// TwinCAT 3 PLC project mobject_core
// Title: mobject-core
// Company: mobject
// Author: mobject dev team
// ProjectVersion: 0.10.0
// ProgramVersion: 3.1.4026.22
// libraries:
//   Tc2_Standard, * (Beckhoff Automation GmbH)
//   Tc2_System, * (Beckhoff Automation GmbH)
//   Tc2_Utilities, * (Beckhoff Automation GmbH)
//   Tc3_JsonXml, * (Beckhoff Automation GmbH)
// project tree:
//   mobject-collections/Dictionary/ Dictionary.TcPOU
//   mobject-collections/Interfaces/Collections/Events/ I_CollectionChangedEvent.TcIO, I_CollectionDisposedEvent.TcIO
//   mobject-collections/Interfaces/Collections/ I_Collection.TcIO (not stored), I_LinkedList.TcIO (not stored), I_List.TcIO, I_Queue.TcIO, I_Stack.TcIO (not stored)
//   mobject-collections/Interfaces/Collections/Nodes/ I_CollectionNode.TcIO, I_LinkedListNode.TcIO, I_ListNode.TcIO
//   mobject-collections/Interfaces/KeyValueCollections/Events/ I_KeyValueCollectionChangedEvent.TcIO, I_KeyValueCollectionDisposedEvent.TcIO
//   mobject-collections/Interfaces/KeyValueCollections/ I_Dictionary.TcIO, I_KeyValueCollection.TcIO
//   mobject-collections/Interfaces/KeyValueCollections/Nodes/ I_DictionaryTreeNode.TcIO (not stored), I_OrderedDictionaryTreeNode.TcIO (not stored)
//   mobject-collections/LinkedList/ LinkedList.TcPOU (not stored)
//   mobject-collections/OrderedDictionary/ OrderedDictionary.TcPOU
//   mobject-collections/Queue/ Queue.TcPOU
//   mobject-collections/Stack/ Stack.TcPOU (not stored)
//   mobject-collections/_Internal/Dictionary/Enumerator/ DictionaryForwardEnumerator.TcPOU (not stored)
//   mobject-collections/_Internal/Dictionary/Node/ DictionaryTreeNode.TcPOU (not stored)
//   mobject-collections/_Internal/Events/Collection/ CollectionChangedEvent.TcPOU, CollectionDisposedEvent.TcPOU, CollectionEvent.TcPOU
//   mobject-collections/_Internal/Events/KeyValueCollection/ KeyValueCollectionChangedEvent.TcPOU (not stored), KeyValueCollectionDisposedEvent.TcPOU (not stored), KeyValueCollectionEvent.TcPOU (not stored)
//   mobject-collections/_Internal/LinkedList/Enumerator/ LinkedListForwardEnumerator.TcPOU (not stored)
//   mobject-collections/_Internal/LinkedList/Node/ LinkedListNode.TcPOU (not stored)
//   mobject-collections/_Internal/OrderedDictionary/Enumerator/ OrderedDictionaryForwardEnumerator.TcPOU
//   mobject-collections/_Internal/OrderedDictionary/Node/ OrderedDictionaryTreeNode.TcPOU
//   mobject-commands/AsyncCommand/ AsyncCommand.TcPOU
//   mobject-commands/AsyncCommand/Interface/ I_AsyncCommand.TcIO (not stored)
//   mobject-commands/AsyncCommand/Runners/ SingleAsyncCommandRunner.TcPOU
//   mobject-commands/Command/Interface/ I_Command.TcIO (not stored)
//   mobject-commands/_Internal/AsyncCommandStateMachine/ AsyncCommandStateMachine.TcPOU (not stored), I_AsyncCommandStateControl.TcIO
//   mobject-constants/ DatatypeLimits.TcGVL (not stored)
//   mobject-converters/Converters/BOOL_TO_/ TryConvert_BOOL_TO_BOOL.TcPOU, TryConvert_BOOL_TO_BYTE.TcPOU (not stored), TryConvert_BOOL_TO_DATE.TcPOU (not stored), TryConvert_BOOL_TO_Destination.TcPOU (not stored), TryConvert_BOOL_TO_DINT.TcPOU (not stored), TryConvert_BOOL_TO_DT.TcPOU, TryConvert_BOOL_TO_DWORD.TcPOU, TryConvert_BOOL_TO_INT.TcPOU (not stored), TryConvert_BOOL_TO_LINT.TcPOU (not stored), TryConvert_BOOL_TO_LREAL.TcPOU, TryConvert_BOOL_TO_LWORD.TcPOU, TryConvert_BOOL_TO_REAL.TcPOU (not stored), TryConvert_BOOL_TO_SINT.TcPOU, TryConvert_BOOL_TO_STRING.TcPOU, TryConvert_BOOL_TO_TIME.TcPOU, TryConvert_BOOL_TO_TOD.TcPOU, TryConvert_BOOL_TO_UDINT.TcPOU (not stored), TryConvert_BOOL_TO_UINT.TcPOU (not stored), TryConvert_BOOL_TO_ULINT.TcPOU (not stored), TryConvert_BOOL_TO_USINT.TcPOU (not stored), TryConvert_BOOL_TO_WORD.TcPOU
//   mobject-converters/Converters/BYTE_TO_/ TryConvert_BYTE_TO_BOOL.TcPOU (not stored), TryConvert_BYTE_TO_BYTE.TcPOU, TryConvert_BYTE_TO_DATE.TcPOU (not stored), TryConvert_BYTE_TO_Destination.TcPOU, TryConvert_BYTE_TO_DINT.TcPOU (not stored), TryConvert_BYTE_TO_DT.TcPOU, TryConvert_BYTE_TO_DWORD.TcPOU (not stored), TryConvert_BYTE_TO_INT.TcPOU (not stored), TryConvert_BYTE_TO_LINT.TcPOU, TryConvert_BYTE_TO_LREAL.TcPOU, TryConvert_BYTE_TO_LWORD.TcPOU, TryConvert_BYTE_TO_REAL.TcPOU (not stored), TryConvert_BYTE_TO_SINT.TcPOU (not stored), TryConvert_BYTE_TO_STRING.TcPOU (not stored), TryConvert_BYTE_TO_TIME.TcPOU (not stored), TryConvert_BYTE_TO_TOD.TcPOU (not stored), TryConvert_BYTE_TO_UDINT.TcPOU, TryConvert_BYTE_TO_UINT.TcPOU, TryConvert_BYTE_TO_ULINT.TcPOU (not stored), TryConvert_BYTE_TO_USINT.TcPOU (not stored), TryConvert_BYTE_TO_WORD.TcPOU (not stored)
//   mobject-converters/Converters/DATE_TO_/ TryConvert_DATE_TO_BOOL.TcPOU, TryConvert_DATE_TO_BYTE.TcPOU, TryConvert_DATE_TO_DATE.TcPOU (not stored), TryConvert_DATE_TO_Destination.TcPOU, TryConvert_DATE_TO_DINT.TcPOU, TryConvert_DATE_TO_DT.TcPOU (not stored), TryConvert_DATE_TO_DWORD.TcPOU (not stored), TryConvert_DATE_TO_INT.TcPOU, TryConvert_DATE_TO_LINT.TcPOU, TryConvert_DATE_TO_LREAL.TcPOU (not stored), TryConvert_DATE_TO_LWORD.TcPOU (not stored), TryConvert_DATE_TO_REAL.TcPOU (not stored), TryConvert_DATE_TO_SINT.TcPOU, TryConvert_DATE_TO_STRING.TcPOU (not stored), TryConvert_DATE_TO_TIME.TcPOU, TryConvert_DATE_TO_TOD.TcPOU (not stored), TryConvert_DATE_TO_UDINT.TcPOU, TryConvert_DATE_TO_UINT.TcPOU (not stored), TryConvert_DATE_TO_ULINT.TcPOU (not stored), TryConvert_DATE_TO_USINT.TcPOU (not stored), TryConvert_DATE_TO_WORD.TcPOU (not stored)
//   mobject-converters/Converters/DINT_TO_/ TryConvert_DINT_TO_BOOL.TcPOU, TryConvert_DINT_TO_BYTE.TcPOU, TryConvert_DINT_TO_DATE.TcPOU (not stored), TryConvert_DINT_TO_Destination.TcPOU (not stored), TryConvert_DINT_TO_DINT.TcPOU (not stored), TryConvert_DINT_TO_DT.TcPOU, TryConvert_DINT_TO_DWORD.TcPOU, TryConvert_DINT_TO_INT.TcPOU, TryConvert_DINT_TO_LINT.TcPOU, TryConvert_DINT_TO_LREAL.TcPOU, TryConvert_DINT_TO_LWORD.TcPOU (not stored), TryConvert_DINT_TO_REAL.TcPOU (not stored), TryConvert_DINT_TO_SINT.TcPOU (not stored), TryConvert_DINT_TO_STRING.TcPOU, TryConvert_DINT_TO_TIME.TcPOU, TryConvert_DINT_TO_TOD.TcPOU, TryConvert_DINT_TO_UDINT.TcPOU (not stored), TryConvert_DINT_TO_UINT.TcPOU, TryConvert_DINT_TO_ULINT.TcPOU (not stored), TryConvert_DINT_TO_USINT.TcPOU, TryConvert_DINT_TO_WORD.TcPOU
//   mobject-converters/Converters/DT_TO_/ TryConvert_DT_TO_BOOL.TcPOU, TryConvert_DT_TO_BYTE.TcPOU, TryConvert_DT_TO_DATE.TcPOU (not stored), TryConvert_DT_TO_Destination.TcPOU (not stored), TryConvert_DT_TO_DINT.TcPOU, TryConvert_DT_TO_DT.TcPOU, TryConvert_DT_TO_DWORD.TcPOU, TryConvert_DT_TO_INT.TcPOU (not stored), TryConvert_DT_TO_LINT.TcPOU, TryConvert_DT_TO_LREAL.TcPOU (not stored), TryConvert_DT_TO_LWORD.TcPOU, TryConvert_DT_TO_REAL.TcPOU, TryConvert_DT_TO_SINT.TcPOU (not stored), TryConvert_DT_TO_STRING.TcPOU (not stored), TryConvert_DT_TO_TIME.TcPOU (not stored), TryConvert_DT_TO_TOD.TcPOU, TryConvert_DT_TO_UDINT.TcPOU (not stored), TryConvert_DT_TO_UINT.TcPOU, TryConvert_DT_TO_ULINT.TcPOU, TryConvert_DT_TO_USINT.TcPOU (not stored), TryConvert_DT_TO_WORD.TcPOU (not stored)
//   mobject-converters/Converters/DWORD_TO_/ TryConvert_DWORD_TO_BOOL.TcPOU (not stored), TryConvert_DWORD_TO_BYTE.TcPOU, TryConvert_DWORD_TO_DATE.TcPOU, TryConvert_DWORD_TO_Destination.TcPOU, TryConvert_DWORD_TO_DINT.TcPOU, TryConvert_DWORD_TO_DT.TcPOU, TryConvert_DWORD_TO_DWORD.TcPOU, TryConvert_DWORD_TO_INT.TcPOU, TryConvert_DWORD_TO_LINT.TcPOU, TryConvert_DWORD_TO_LREAL.TcPOU (not stored), TryConvert_DWORD_TO_LWORD.TcPOU, TryConvert_DWORD_TO_REAL.TcPOU, TryConvert_DWORD_TO_SINT.TcPOU (not stored), TryConvert_DWORD_TO_STRING.TcPOU, TryConvert_DWORD_TO_TIME.TcPOU, TryConvert_DWORD_TO_TOD.TcPOU, TryConvert_DWORD_TO_UDINT.TcPOU (not stored), TryConvert_DWORD_TO_UINT.TcPOU (not stored), TryConvert_DWORD_TO_ULINT.TcPOU (not stored), TryConvert_DWORD_TO_USINT.TcPOU, TryConvert_DWORD_TO_WORD.TcPOU (not stored)
//   mobject-converters/Converters/INT_TO_/ TryConvert_INT_TO_BOOL.TcPOU (not stored), TryConvert_INT_TO_BYTE.TcPOU (not stored), TryConvert_INT_TO_DATE.TcPOU, TryConvert_INT_TO_Destination.TcPOU (not stored), TryConvert_INT_TO_DINT.TcPOU (not stored), TryConvert_INT_TO_DT.TcPOU, TryConvert_INT_TO_DWORD.TcPOU (not stored), TryConvert_INT_TO_INT.TcPOU, TryConvert_INT_TO_LINT.TcPOU, TryConvert_INT_TO_LREAL.TcPOU (not stored), TryConvert_INT_TO_LWORD.TcPOU, TryConvert_INT_TO_REAL.TcPOU, TryConvert_INT_TO_SINT.TcPOU (not stored), TryConvert_INT_TO_STRING.TcPOU, TryConvert_INT_TO_TIME.TcPOU, TryConvert_INT_TO_TOD.TcPOU (not stored), TryConvert_INT_TO_UDINT.TcPOU, TryConvert_INT_TO_UINT.TcPOU (not stored), TryConvert_INT_TO_ULINT.TcPOU, TryConvert_INT_TO_USINT.TcPOU, TryConvert_INT_TO_WORD.TcPOU
//   mobject-converters/Converters/LINT_TO_/ TryConvert_LINT_TO_BOOL.TcPOU, TryConvert_LINT_TO_BYTE.TcPOU, TryConvert_LINT_TO_DATE.TcPOU, TryConvert_LINT_TO_Destination.TcPOU (not stored), TryConvert_LINT_TO_DINT.TcPOU, TryConvert_LINT_TO_DT.TcPOU, TryConvert_LINT_TO_DWORD.TcPOU, TryConvert_LINT_TO_INT.TcPOU, TryConvert_LINT_TO_LINT.TcPOU, TryConvert_LINT_TO_LREAL.TcPOU, TryConvert_LINT_TO_LWORD.TcPOU (not stored), TryConvert_LINT_TO_REAL.TcPOU (not stored), TryConvert_LINT_TO_SINT.TcPOU (not stored), TryConvert_LINT_TO_STRING.TcPOU, TryConvert_LINT_TO_TIME.TcPOU, TryConvert_LINT_TO_TOD.TcPOU, TryConvert_LINT_TO_UDINT.TcPOU (not stored), TryConvert_LINT_TO_UINT.TcPOU, TryConvert_LINT_TO_ULINT.TcPOU, TryConvert_LINT_TO_USINT.TcPOU, TryConvert_LINT_TO_WORD.TcPOU (not stored)
//   mobject-converters/Converters/LREAL_TO_/ TryConvert_LREAL_TO_BOOL.TcPOU, TryConvert_LREAL_TO_BYTE.TcPOU (not stored), TryConvert_LREAL_TO_DATE.TcPOU, TryConvert_LREAL_TO_Destination.TcPOU (not stored), TryConvert_LREAL_TO_DINT.TcPOU (not stored), TryConvert_LREAL_TO_DT.TcPOU, TryConvert_LREAL_TO_DWORD.TcPOU (not stored), TryConvert_LREAL_TO_INT.TcPOU, TryConvert_LREAL_TO_LINT.TcPOU (not stored), TryConvert_LREAL_TO_LREAL.TcPOU (not stored), TryConvert_LREAL_TO_LWORD.TcPOU (not stored), TryConvert_LREAL_TO_REAL.TcPOU (not stored), TryConvert_LREAL_TO_SINT.TcPOU (not stored), TryConvert_LREAL_TO_STRING.TcPOU, TryConvert_LREAL_TO_TIME.TcPOU (not stored), TryConvert_LREAL_TO_TOD.TcPOU (not stored), TryConvert_LREAL_TO_UDINT.TcPOU (not stored), TryConvert_LREAL_TO_UINT.TcPOU, TryConvert_LREAL_TO_ULINT.TcPOU, TryConvert_LREAL_TO_USINT.TcPOU, TryConvert_LREAL_TO_WORD.TcPOU
//   mobject-converters/Converters/LWORD_TO_/ TryConvert_LWORD_TO_BOOL.TcPOU (not stored), TryConvert_LWORD_TO_BYTE.TcPOU, TryConvert_LWORD_TO_DATE.TcPOU, TryConvert_LWORD_TO_Destination.TcPOU (not stored), TryConvert_LWORD_TO_DINT.TcPOU (not stored), TryConvert_LWORD_TO_DT.TcPOU (not stored), TryConvert_LWORD_TO_DWORD.TcPOU, TryConvert_LWORD_TO_INT.TcPOU, TryConvert_LWORD_TO_LINT.TcPOU (not stored), TryConvert_LWORD_TO_LREAL.TcPOU (not stored), TryConvert_LWORD_TO_LWORD.TcPOU, TryConvert_LWORD_TO_REAL.TcPOU, TryConvert_LWORD_TO_SINT.TcPOU, TryConvert_LWORD_TO_STRING.TcPOU (not stored), TryConvert_LWORD_TO_TIME.TcPOU (not stored), TryConvert_LWORD_TO_TOD.TcPOU (not stored), TryConvert_LWORD_TO_UDINT.TcPOU (not stored), TryConvert_LWORD_TO_UINT.TcPOU (not stored), TryConvert_LWORD_TO_ULINT.TcPOU, TryConvert_LWORD_TO_USINT.TcPOU (not stored), TryConvert_LWORD_TO_WORD.TcPOU
//   mobject-converters/Converters/REAL_TO_/ TryConvert_REAL_TO_BOOL.TcPOU (not stored), TryConvert_REAL_TO_BYTE.TcPOU (not stored), TryConvert_REAL_TO_DATE.TcPOU, TryConvert_REAL_TO_Destination.TcPOU (not stored), TryConvert_REAL_TO_DINT.TcPOU, TryConvert_REAL_TO_DT.TcPOU, TryConvert_REAL_TO_DWORD.TcPOU, TryConvert_REAL_TO_INT.TcPOU, TryConvert_REAL_TO_LINT.TcPOU, TryConvert_REAL_TO_LREAL.TcPOU (not stored), TryConvert_REAL_TO_LWORD.TcPOU (not stored), TryConvert_REAL_TO_REAL.TcPOU, TryConvert_REAL_TO_SINT.TcPOU, TryConvert_REAL_TO_STRING.TcPOU, TryConvert_REAL_TO_TIME.TcPOU, TryConvert_REAL_TO_TOD.TcPOU, TryConvert_REAL_TO_UDINT.TcPOU, TryConvert_REAL_TO_UINT.TcPOU, TryConvert_REAL_TO_ULINT.TcPOU, TryConvert_REAL_TO_USINT.TcPOU, TryConvert_REAL_TO_WORD.TcPOU
//   mobject-converters/Converters/SINT_TO_/ TryConvert_SINT_TO_BOOL.TcPOU (not stored), TryConvert_SINT_TO_BYTE.TcPOU, TryConvert_SINT_TO_DATE.TcPOU (not stored), TryConvert_SINT_TO_Destination.TcPOU (not stored), TryConvert_SINT_TO_DINT.TcPOU (not stored), TryConvert_SINT_TO_DT.TcPOU, TryConvert_SINT_TO_DWORD.TcPOU (not stored), TryConvert_SINT_TO_INT.TcPOU, TryConvert_SINT_TO_LINT.TcPOU, TryConvert_SINT_TO_LREAL.TcPOU, TryConvert_SINT_TO_LWORD.TcPOU (not stored), TryConvert_SINT_TO_REAL.TcPOU (not stored), TryConvert_SINT_TO_SINT.TcPOU (not stored), TryConvert_SINT_TO_STRING.TcPOU (not stored), TryConvert_SINT_TO_TIME.TcPOU (not stored), TryConvert_SINT_TO_TOD.TcPOU (not stored), TryConvert_SINT_TO_UDINT.TcPOU, TryConvert_SINT_TO_UINT.TcPOU, TryConvert_SINT_TO_ULINT.TcPOU, TryConvert_SINT_TO_USINT.TcPOU (not stored), TryConvert_SINT_TO_WORD.TcPOU (not stored)
//   mobject-converters/Converters/STRING_TO_/ TryConvert_STRING_TO_BOOL.TcPOU (not stored), TryConvert_STRING_TO_BYTE.TcPOU, TryConvert_STRING_TO_DATE.TcPOU, TryConvert_STRING_TO_Destination.TcPOU, TryConvert_STRING_TO_DINT.TcPOU, TryConvert_STRING_TO_DT.TcPOU (not stored), TryConvert_STRING_TO_DWORD.TcPOU, TryConvert_STRING_TO_INT.TcPOU (not stored), TryConvert_STRING_TO_LINT.TcPOU (not stored), TryConvert_STRING_TO_LREAL.TcPOU, TryConvert_STRING_TO_LWORD.TcPOU (not stored), TryConvert_STRING_TO_REAL.TcPOU, TryConvert_STRING_TO_SINT.TcPOU, TryConvert_STRING_TO_STRING.TcPOU, TryConvert_STRING_TO_TIME.TcPOU (not stored), TryConvert_STRING_TO_TOD.TcPOU, TryConvert_STRING_TO_UDINT.TcPOU (not stored), TryConvert_STRING_TO_UINT.TcPOU, TryConvert_STRING_TO_ULINT.TcPOU, TryConvert_STRING_TO_USINT.TcPOU, TryConvert_STRING_TO_WORD.TcPOU
//   mobject-converters/Converters/TIME_TO_/ TryConvert_TIME_TO_BOOL.TcPOU, TryConvert_TIME_TO_BYTE.TcPOU, TryConvert_TIME_TO_DATE.TcPOU (not stored), TryConvert_TIME_TO_Destination.TcPOU (not stored), TryConvert_TIME_TO_DINT.TcPOU, TryConvert_TIME_TO_DT.TcPOU (not stored), TryConvert_TIME_TO_DWORD.TcPOU, TryConvert_TIME_TO_INT.TcPOU, TryConvert_TIME_TO_LINT.TcPOU (not stored), TryConvert_TIME_TO_LREAL.TcPOU (not stored), TryConvert_TIME_TO_LWORD.TcPOU, TryConvert_TIME_TO_REAL.TcPOU, TryConvert_TIME_TO_SINT.TcPOU, TryConvert_TIME_TO_STRING.TcPOU, TryConvert_TIME_TO_TIME.TcPOU, TryConvert_TIME_TO_TOD.TcPOU (not stored), TryConvert_TIME_TO_UDINT.TcPOU, TryConvert_TIME_TO_UINT.TcPOU (not stored), TryConvert_TIME_TO_ULINT.TcPOU (not stored), TryConvert_TIME_TO_USINT.TcPOU, TryConvert_TIME_TO_WORD.TcPOU
//   mobject-converters/Converters/TOD_TO_/ TryConvert_TOD_TO_BOOL.TcPOU, TryConvert_TOD_TO_BYTE.TcPOU, TryConvert_TOD_TO_DATE.TcPOU (not stored), TryConvert_TOD_TO_Destination.TcPOU, TryConvert_TOD_TO_DINT.TcPOU (not stored), TryConvert_TOD_TO_DT.TcPOU (not stored), TryConvert_TOD_TO_DWORD.TcPOU (not stored), TryConvert_TOD_TO_INT.TcPOU, TryConvert_TOD_TO_LINT.TcPOU, TryConvert_TOD_TO_LREAL.TcPOU (not stored), TryConvert_TOD_TO_LWORD.TcPOU (not stored), TryConvert_TOD_TO_REAL.TcPOU, TryConvert_TOD_TO_SINT.TcPOU (not stored), TryConvert_TOD_TO_STRING.TcPOU (not stored), TryConvert_TOD_TO_TIME.TcPOU, TryConvert_TOD_TO_TOD.TcPOU (not stored), TryConvert_TOD_TO_UDINT.TcPOU (not stored), TryConvert_TOD_TO_UINT.TcPOU (not stored), TryConvert_TOD_TO_ULINT.TcPOU (not stored), TryConvert_TOD_TO_USINT.TcPOU, TryConvert_TOD_TO_WORD.TcPOU
//   mobject-converters/Converters/ TryConvert_Source_TO_Destination.TcPOU (not stored)
//   mobject-converters/Converters/UDINT_TO_/ TryConvert_UDINT_TO_BOOL.TcPOU, TryConvert_UDINT_TO_BYTE.TcPOU, TryConvert_UDINT_TO_DATE.TcPOU, TryConvert_UDINT_TO_Destination.TcPOU (not stored), TryConvert_UDINT_TO_DINT.TcPOU (not stored), TryConvert_UDINT_TO_DT.TcPOU (not stored), TryConvert_UDINT_TO_DWORD.TcPOU, TryConvert_UDINT_TO_INT.TcPOU, TryConvert_UDINT_TO_LINT.TcPOU (not stored), TryConvert_UDINT_TO_LREAL.TcPOU, TryConvert_UDINT_TO_LWORD.TcPOU, TryConvert_UDINT_TO_REAL.TcPOU, TryConvert_UDINT_TO_SINT.TcPOU (not stored), TryConvert_UDINT_TO_STRING.TcPOU, TryConvert_UDINT_TO_TIME.TcPOU (not stored), TryConvert_UDINT_TO_TOD.TcPOU (not stored), TryConvert_UDINT_TO_UDINT.TcPOU (not stored), TryConvert_UDINT_TO_UINT.TcPOU (not stored), TryConvert_UDINT_TO_ULINT.TcPOU (not stored), TryConvert_UDINT_TO_USINT.TcPOU, TryConvert_UDINT_TO_WORD.TcPOU
//   mobject-converters/Converters/UINT_TO_/ TryConvert_UINT_TO_BOOL.TcPOU, TryConvert_UINT_TO_BYTE.TcPOU (not stored), TryConvert_UINT_TO_DATE.TcPOU, TryConvert_UINT_TO_Destination.TcPOU, TryConvert_UINT_TO_DINT.TcPOU (not stored), TryConvert_UINT_TO_DT.TcPOU (not stored), TryConvert_UINT_TO_DWORD.TcPOU, TryConvert_UINT_TO_INT.TcPOU, TryConvert_UINT_TO_LINT.TcPOU, TryConvert_UINT_TO_LREAL.TcPOU, TryConvert_UINT_TO_LWORD.TcPOU (not stored), TryConvert_UINT_TO_REAL.TcPOU, TryConvert_UINT_TO_SINT.TcPOU, TryConvert_UINT_TO_STRING.TcPOU (not stored), TryConvert_UINT_TO_TIME.TcPOU, TryConvert_UINT_TO_TOD.TcPOU, TryConvert_UINT_TO_UDINT.TcPOU, TryConvert_UINT_TO_UINT.TcPOU, TryConvert_UINT_TO_ULINT.TcPOU (not stored), TryConvert_UINT_TO_USINT.TcPOU (not stored), TryConvert_UINT_TO_WORD.TcPOU (not stored)
//   mobject-converters/Converters/ULINT_TO_/ TryConvert_ULINT_TO_BOOL.TcPOU (not stored), TryConvert_ULINT_TO_BYTE.TcPOU, TryConvert_ULINT_TO_DATE.TcPOU, TryConvert_ULINT_TO_Destination.TcPOU, TryConvert_ULINT_TO_DINT.TcPOU (not stored), TryConvert_ULINT_TO_DT.TcPOU (not stored), TryConvert_ULINT_TO_DWORD.TcPOU, TryConvert_ULINT_TO_INT.TcPOU, TryConvert_ULINT_TO_LINT.TcPOU, TryConvert_ULINT_TO_LREAL.TcPOU, TryConvert_ULINT_TO_LWORD.TcPOU (not stored), TryConvert_ULINT_TO_REAL.TcPOU, TryConvert_ULINT_TO_SINT.TcPOU (not stored), TryConvert_ULINT_TO_STRING.TcPOU (not stored), TryConvert_ULINT_TO_TIME.TcPOU, TryConvert_ULINT_TO_TOD.TcPOU, TryConvert_ULINT_TO_UDINT.TcPOU (not stored), TryConvert_ULINT_TO_UINT.TcPOU, TryConvert_ULINT_TO_ULINT.TcPOU, TryConvert_ULINT_TO_USINT.TcPOU (not stored), TryConvert_ULINT_TO_WORD.TcPOU
//   mobject-converters/Converters/USINT_TO_/ TryConvert_USINT_TO_BOOL.TcPOU (not stored), TryConvert_USINT_TO_BYTE.TcPOU (not stored), TryConvert_USINT_TO_DATE.TcPOU, TryConvert_USINT_TO_Destination.TcPOU, TryConvert_USINT_TO_DINT.TcPOU (not stored), TryConvert_USINT_TO_DT.TcPOU (not stored), TryConvert_USINT_TO_DWORD.TcPOU, TryConvert_USINT_TO_INT.TcPOU (not stored), TryConvert_USINT_TO_LINT.TcPOU, TryConvert_USINT_TO_LREAL.TcPOU, TryConvert_USINT_TO_LWORD.TcPOU (not stored), TryConvert_USINT_TO_REAL.TcPOU, TryConvert_USINT_TO_SINT.TcPOU, TryConvert_USINT_TO_STRING.TcPOU, TryConvert_USINT_TO_TIME.TcPOU, TryConvert_USINT_TO_TOD.TcPOU (not stored), TryConvert_USINT_TO_UDINT.TcPOU, TryConvert_USINT_TO_UINT.TcPOU (not stored), TryConvert_USINT_TO_ULINT.TcPOU (not stored), TryConvert_USINT_TO_USINT.TcPOU, TryConvert_USINT_TO_WORD.TcPOU
//   mobject-converters/Converters/WORD_TO_/ TryConvert_WORD_TO_BOOL.TcPOU (not stored), TryConvert_WORD_TO_BYTE.TcPOU, TryConvert_WORD_TO_DATE.TcPOU, TryConvert_WORD_TO_Destination.TcPOU, TryConvert_WORD_TO_DINT.TcPOU, TryConvert_WORD_TO_DT.TcPOU (not stored), TryConvert_WORD_TO_DWORD.TcPOU, TryConvert_WORD_TO_INT.TcPOU, TryConvert_WORD_TO_LINT.TcPOU (not stored), TryConvert_WORD_TO_LREAL.TcPOU, TryConvert_WORD_TO_LWORD.TcPOU (not stored), TryConvert_WORD_TO_REAL.TcPOU (not stored), TryConvert_WORD_TO_SINT.TcPOU (not stored), TryConvert_WORD_TO_STRING.TcPOU, TryConvert_WORD_TO_TIME.TcPOU (not stored), TryConvert_WORD_TO_TOD.TcPOU, TryConvert_WORD_TO_UDINT.TcPOU, TryConvert_WORD_TO_UINT.TcPOU, TryConvert_WORD_TO_ULINT.TcPOU (not stored), TryConvert_WORD_TO_USINT.TcPOU (not stored), TryConvert_WORD_TO_WORD.TcPOU
//   mobject-datatypes/DatatypeOperations/Collection/ DatatypeOperations.TcPOU
//   mobject-datatypes/DatatypeOperations/Interface/ I_DatatypeOperation.TcIO (not stored)
//   mobject-datatypes/DatatypeOperations/ MemCopyOperation.TcPOU (not stored), SafeMemCopyOperation.TcPOU (not stored), WriteBitToBoolOperation.TcPOU, WriteBoolToBitOperation.TcPOU
//   mobject-datatypes/Datatypes/Base/ Datatypes.TcPOU (not stored)
//   mobject-datatypes/Datatypes/Events/ I_AliasDatatypeAddedEvent.TcIO (not stored), I_DatatypeAddedEvent.TcIO, I_EnumDatatypeAddedEvent.TcIO, I_InterfaceDatatypeAddedEvent.TcIO (not stored), I_StructuredDatatypeAddedEvent.TcIO (not stored), I_ArrayDatatypeAddedEvent.TcIO (not stored)
//   mobject-datatypes/Datatypes/Interface/ I_Datatypes.TcIO
//   mobject-datatypes/DatatypeVisitor/ I_DatatypeVisitor.TcIO
//   mobject-datatypes/Functions/ GetByteOffset.TcPOU (not stored)
//   mobject-datatypes/Primitive/Interfaces/ I_BIT.TcIO, I_BYTE.TcIO, I_ANY.TcIO, I_DINT.TcIO, I_DT.TcIO, I_DWORD.TcIO, I_INT.TcIO, I_LINT.TcIO, I_LREAL.TcIO, I_LWORD.TcIO, I_PVOID.TcIO, I_REAL.TcIO, I_REFERENCE_TO.TcIO, I_SINT.TcIO, I_TOD.TcIO, I_TIME_OF_DAY.TcIO, I_STRING.TcIO, I_BOOL.TcIO, I_UDINT.TcIO, I_UINT.TcIO, I_ULINT.TcIO, I_USINT.TcIO, I_WORD.TcIO
//   mobject-datatypes/Primitive/ _REFERENCE_TO.TcPOU, _NULL.TcPOU, _BIT.TcPOU, _BOOL.TcPOU, _ANY.TcPOU, _BYTE.TcPOU, _DINT.TcPOU, _DT.TcPOU, _DWORD.TcPOU, _INT.TcPOU, _LINT.TcPOU, _LREAL.TcPOU, _LWORD.TcPOU, _REAL.TcPOU, _SINT.TcPOU, _STRING.TcPOU, _TIME_OF_DAY.TcPOU, _TOD.TcPOU, _UDINT.TcPOU, _PVOID.TcPOU, _UINT.TcPOU, _ULINT.TcPOU, _USINT.TcPOU, _WORD.TcPOU
//   mobject-datatypes/_Internal/Datatype/ AliasDatatypeBase.TcPOU, ArrayDatatypeBase_2D.TcPOU (not stored), ArrayDatatypeBase_3D.TcPOU, DatatypeBase.TcPOU, EnumDatatypeBase.TcPOU, InterfaceDatatypeBase.TcPOU, NumericDatatypeBase.TcPOU (not stored), StructuredDatatypeBase.TcPOU, ArrayDatatypeBase_1D.TcPOU (not stored), UserDefinedDatatypeBase.TcPOU
//   mobject-datatypes/_Internal/Datatype/Interface/ I_AliasDatatype.TcIO, I_ArrayDatatype_1D.TcIO, I_ArrayDatatype_2D.TcIO (not stored), I_ArrayDatatype_3D.TcIO, I_Datatype.TcIO, I_EnumDatatype.TcIO, I_InterfaceDatatype.TcIO, I_NumericDatatype.TcIO (not stored), I_StructuredDatatype.TcIO, I_ArrayDatatype.TcIO, I_UserDefinedDatatype.TcIO
//   mobject-datatypes/_Internal/Errors/ UnknownEnumerationError.TcPOU (not stored)
//   mobject-datatypes/_Internal/Events/ AliasDatatypeAddedEvent.TcPOU (not stored), DatatypeAddedEvent.TcPOU, EnumDatatypeAddedEvent.TcPOU (not stored), InterfaceDatatypeAddedEvent.TcPOU, StructuredDatatypeAddedEvent.TcPOU, ArrayDatatypeAddedEvent.TcPOU (not stored)
//   mobject-datatypes/_Internal/StructureMembers/Host/ StructureMemberHost.TcPOU
//   mobject-datatypes/_Internal/StructureMembers/Interface/ I_HostStructureMembers.TcIO, I_StructureMembers.TcIO (not stored)
//   mobject-deserialization/DeserializationFeedback/ DeserializerFeedback.TcPOU
//   mobject-deserialization/Errors/CustomError/ CustomDeserializationFailedError.TcPOU (not stored)
//   mobject-deserialization/Errors/ DeserializationErrorFactory.TcPOU
//   mobject-deserialization/Errors/IncorrectType/ IncorrectKeyTypeDeserializationError.TcPOU, IncorrectTypeDeserializationError.TcPOU
//   mobject-deserialization/Errors/Invalid Index/ InvalidArrayIndexDeserializationError.TcPOU
//   mobject-deserialization/Errors/Invalid Key/ InvalidKeyDeserializationError.TcPOU (not stored)
//   mobject-deserialization/Errors/Missing Key/ MissingKeyDeserializationError.TcPOU
//   mobject-deserialization/GarbageCollector/ DeserializerGarbageCollector.TcPOU, I_DeserializerGarbageCollector.TcIO (not stored)
//   mobject-deserialization/Interfaces/ I_Deserializable.TcIO (not stored), I_Deserializer.TcIO, I_DeserializerArrayForwardEnumerator.TcIO, I_DeserializerFeedback.TcIO, I_DeserializerObjectForwardEnumerator.TcIO
//   mobject-errors/Errors/ Error.TcPOU (not stored), NullError.TcPOU
//   mobject-errors/Interfaces/ I_Error.TcIO, I_ErrorVisitor.TcIO
//   mobject-events/EventEmitter/ EventEmitter.TcPOU (not stored)
//   mobject-events/Interfaces/ I_Event.TcIO, I_EventEmitter.TcIO (not stored), I_EventHandler.TcIO (not stored), I_EventTarget.TcIO (not stored)
//   mobject-events/_Internal/EventHandlerItem/ EventHandlerItem.TcPOU, EventHandlerItemOnceOnly.TcPOU, I_EventHandlerItem.TcIO
//   mobject-disposable/Disposable/ Disposable.TcPOU (not stored)
//   mobject-disposable/Interfaces/ I_Disposable.TcIO (not stored)
//   mobject-enumerable/Interfaces/Enumerators/ I_ForwardEnumerator.TcIO, I_KeyValueForwardEnumerator.TcIO (not stored)
//   mobject-enumerable/Interfaces/ I_Enumerable.TcIO, I_KeyValueEnumerable.TcIO
//   mobject-json/JsonDeserializer/Events/ I_JsonDeserializerChangedEvent.TcIO (not stored), I_JsonDeserializerDisposedEvent.TcIO
//   mobject-json/JsonDeserializer/ I_JsonDeserializer.TcIO, JsonDeserializer.TcPOU
//   mobject-json/JsonDomParser/ JsonDomParser.TcPOU
//   mobject-json/JsonSerializer/ JsonSerializer.TcPOU
//   mobject-json/_Internal/Events/ JsonDeserializerChangedEvent.TcPOU, JsonDeserializerDisposedEvent.TcPOU (not stored), JsonDeserializerEvent.TcPOU
//   mobject-json/_Internal/JsonDeserializerForwardEnumerator/ JsonDeserializerArrayForwardEnumerator.TcPOU, JsonDeserializerNullArrayForwardEnumerator.TcPOU, JsonDeserializerNullObjectForwardEnumerator.TcPOU (not stored), JsonDeserializerObjectForwardEnumerator.TcPOU
//   mobject-json/_Internal/JsonDeserializerNode/ JsonDeserializerNode.TcPOU, JsonDeserializerNullNode.TcPOU
//   mobject-json/_Internal/JsonPathSyntaxParser/ JsonPathSyntaxParser.TcPOU
//   mobject-json/_Internal/JsonPathVisitor/ I_JsonPathVisitor.TcIO (not stored), JsonDomCreator.TcPOU, JsonDomNavigator.TcPOU (not stored)
//   mobject-serialization/Interfaces/ I_Serializable.TcIO, I_Serializer.TcIO
//   mobject-server/GVLs/ ServerConfiguration.TcGVL
//   mobject-server/RpcApi/ I_RpcApi.TcIO
//   mobject-server/RpcHandler/Examples/ AsyncConcatStringRpcHandler.TcPOU, ConcatStringRpcHandler.TcPOU
//   mobject-server/RpcHandler/ I_AsynchronousRpcHandler.TcIO, I_SynchronousRpcHandler.TcIO
//   mobject-server/RpcServer/ I_RpcServer.TcIO, RpcServer.TcPOU
//   mobject-server/_Internal/AsyncResponse/HeaderAccessor/ I_AsyncResponseHeaderAccessor.TcIO
//   mobject-server/_Internal/AsyncResponse/Manager/ AsyncResponseManager.TcPOU, I_AsyncResponseManager.TcIO
//   mobject-server/_Internal/AsyncResponse/Middleware/ AsyncResponseMiddleware.TcPOU
//   mobject-server/_Internal/AsyncResponse/Proxy/ AsyncResponseSessionDataProxy.TcPOU
//   mobject-server/_Internal/AsyncResponse/SessionData/ AsyncResponseSessionData.TcPOU, I_AsyncResponseSessionData.TcIO
//   mobject-server/_Internal/ChunkedRequests/ChunkedRequest/ ChunkedRequest.TcPOU
//   mobject-server/_Internal/ChunkedRequests/HeaderAccessor/ I_ChunkedRequestsHeaderAccessor.TcIO
//   mobject-server/_Internal/ChunkedRequests/Manager/ ChunkedRequestsManager.TcPOU, I_ChunkedRequestsManager.TcIO
//   mobject-server/_Internal/ChunkedRequests/Middleware/ ChunkedRequestsMiddleware.TcPOU
//   mobject-server/_Internal/ChunkedRequests/SessionData/ ChunkedRequestData.TcPOU, I_ChunkedRequestData.TcIO
//   mobject-server/_Internal/ChunkedResponses/HeaderAccessor/ I_ChunkedResponseHeaderAccessor.TcIO
//   mobject-server/_Internal/ChunkedResponses/Manager/ ChunkedResponseManager.TcPOU, I_ChunkedResponseManager.TcIO
//   mobject-server/_Internal/ChunkedResponses/Middleware/ ChunkedResponsesMiddleware.TcPOU
//   mobject-server/_Internal/ChunkedResponses/ServerResponse/ ChunkableServerResponse.TcPOU
//   mobject-server/_Internal/ChunkedResponses/SessionData/ ChunkedResponseData.TcPOU, I_ChunkedResponseData.TcIO
//   mobject-server/_Internal/Followup/Middleware/ ResponseIdGuardMiddleware.TcPOU
//   mobject-server/_Internal/HeaderAccessor/ HeaderAccessor.TcPOU
//   mobject-server/_Internal/Header/ Header.TcPOU, I_Header.TcIO
//   mobject-server/_Internal/Middleware/Base/ MiddlewareBase.TcPOU
//   mobject-server/_Internal/Middleware/Interface/ I_Middleware.TcIO
//   mobject-server/_Internal/Middleware/Stack/ MiddlewareStack.TcPOU
//   mobject-server/_Internal/Request/Interface/ I_Request.TcIO
//   mobject-server/_Internal/Request/ Request.TcPOU
//   mobject-server/_Internal/ResponseId/Interface/ I_ResponseIdGenerator.TcIO
//   mobject-server/_Internal/ResponseId/ SequentialResponseIdGenerator.TcPOU
//   mobject-server/_Internal/RPC/AsyncRpcCallQueue/ AsyncRpcCallQueue.TcPOU, I_AsyncRpcCallQueue.TcIO
//   mobject-server/_Internal/RPC/AsyncRpcCall/ AsyncRpcCall.TcPOU, I_AsyncRpcCall.TcIO
//   mobject-server/_Internal/RPC/Handlers/ AsynchronousRpcHandlers.TcPOU, I_AsynchronousRpcHandlers.TcIO, I_HostAsynchronousRpcHandlers.TcIO, I_HostSynchronousRpcHandlers.TcIO, I_SynchronousRpcHandlers.TcIO, SynchronousRpcHandlers.TcPOU
//   mobject-server/_Internal/RPC/HeaderAccessor/ I_RpcHeaderAccessor.TcIO
//   mobject-server/_Internal/RPC/Manager/ I_RpcManager.TcIO, RpcManager.TcPOU
//   mobject-server/_Internal/RPC/Middleware/ RpcMiddleware.TcPOU
//   mobject-server/_Internal/RPC/RegisteredRpcApis/ RegisteredRpcApis.TcPOU
//   mobject-server/_Internal/RPC/Response/Async/ AsynchronousRpcResponse.TcPOU, I_AsynchronousRpcResponse.TcIO
//   mobject-server/_Internal/RPC/Response/Factory/ AsynchronousRpcResponseFactory.TcPOU, I_AsynchronousRpcResponseFactory.TcIO
//   mobject-server/_Internal/RPC/Response/Sync/ I_SynchronousRpcResponse.TcIO, SynchronousRpcResponse.TcPOU
//   mobject-server/_Internal/ServerResponse/Data/ ResponseData.TcDUT
//   mobject-server/_Internal/ServerResponse/HeaderAccessor/ I_ServerResponseHeaderAccessor.TcIO
//   mobject-server/_Internal/ServerResponse/Interface/ I_ServerResponse.TcIO
//   mobject-server/_Internal/ServerResponse/ ServerResponse.TcPOU
//   mobject-server/_Internal/Sessions/HeaderAccessor/ I_SessionHeaderAccessor.TcIO
//   mobject-server/_Internal/Sessions/Manager/ I_SessionManager.TcIO, SessionManager.TcPOU
//   mobject-server/_Internal/Sessions/Middleware/ SessionsMiddleware.TcPOU
//   mobject-server/_Internal/Sessions/SessionData/ I_SessionData.TcIO
//   mobject-server/_Internal/Sessions/SessionId/ I_SessionIdGenerator.TcIO, SequentialSessionIdGenerator.TcPOU
//   mobject-server/_Internal/Sessions/Session/ I_Session.TcIO, Session.TcPOU
//   mobject-server/_Internal/Sessions/Storage/ I_SessionStorage.TcIO
//   mobject-server/_Internal/TimeStamp/ I_Timestamp.TcIO, SystemTimestamp.TcPOU

// ---- mobject-server/_Internal/ServerResponse/Data/ResponseData.TcDUT
TYPE ResponseData : 
STRUCT
	Header : STRING(ServerConfiguration.HEADER_STRING_SIZE);
	Payload : STRING(ServerConfiguration.PAYLOAD_STRING_SIZE);
END_STRUCT
END_TYPE

// ---- mobject-server/GVLs/ServerConfiguration.TcGVL
{attribute 'qualified_only'}
VAR_GLOBAL CONSTANT
	HEADER_STRING_SIZE : UDINT := 1024;
	PAYLOAD_STRING_SIZE : UDINT := 8000; // typically 1/8th of the Runtime Stack Size

	// Maximum time an asynchronous response may remain pending.
    // T#0S disables the deadline.
    PENDING_RESPONSE_MAX_AGE : TIME := T#60S;

    // Delay suggested to clients between asynchronous response polls.
    // Prevents clients continuously polling the PLC as fast as ADS allows.
    PENDING_RESPONSE_RETRY_DELAY_MS : UDINT := 20;
END_VAR

// ---- mobject-collections/Interfaces/Collections/Events/I_CollectionChangedEvent.TcIO
INTERFACE I_CollectionChangedEvent EXTENDS I_Event

PROPERTY PUBLIC Target : I_Collection
GET
END_GET
END_PROPERTY

END_INTERFACE

// ---- mobject-collections/Interfaces/Collections/Events/I_CollectionDisposedEvent.TcIO
INTERFACE I_CollectionDisposedEvent EXTENDS I_Event

PROPERTY PUBLIC Target : I_Collection
GET
END_GET
END_PROPERTY

END_INTERFACE

// ---- mobject-collections/Interfaces/Collections/I_List.TcIO
INTERFACE I_List EXTENDS I_Collection

PROPERTY PUBLIC Capacity : DINT
GET
END_GET
END_PROPERTY

METHOD PUBLIC GetIndexOf : DINT
VAR_INPUT
	Item : ANY;
END_VAR
END_METHOD

METHOD PUBLIC TrimExcess
END_METHOD

METHOD PUBLIC TryGetByIndex : BOOL
VAR_INPUT
	Index : DINT;
	Destination : ANY;
END_VAR
END_METHOD

METHOD PUBLIC TryGetToByIndex : BOOL
VAR_INPUT
	Index : DINT;
	DestinationAddress : PVOID;
	DestinationSize : UDINT;
END_VAR
END_METHOD

METHOD TryInsert : BOOL
VAR_INPUT
	Index : DINT;
	Item : ANY;
END_VAR
END_METHOD

METHOD TryRemoveAt : BOOL
VAR_INPUT
	Index : DINT;
END_VAR
END_METHOD

END_INTERFACE

// ---- mobject-collections/Interfaces/Collections/I_Queue.TcIO
INTERFACE I_Queue EXTENDS I_Collection

METHOD PUBLIC Enqueue
VAR_INPUT
	Item : ANY;
END_VAR
END_METHOD

METHOD PUBLIC TryDequeue : BOOL;
VAR_INPUT
	Destination : ANY;
END_VAR
END_METHOD

METHOD PUBLIC TryPeek : BOOL;
VAR_INPUT
	Destination : ANY;
END_VAR
END_METHOD

END_INTERFACE

// ---- mobject-collections/Interfaces/Collections/Nodes/I_CollectionNode.TcIO
INTERFACE I_CollectionNode EXTENDS I_Disposable

PROPERTY PUBLIC DataSize : UDINT
GET
END_GET
END_PROPERTY

METHOD PUBLIC Equals : BOOL
VAR_INPUT
	Symbol : ANY;
END_VAR
END_METHOD

METHOD PUBLIC TryGet : BOOL;
VAR_INPUT
	Destination : ANY;
END_VAR
END_METHOD

METHOD PUBLIC TryGetTo : BOOL;
VAR_INPUT
	DestinationAddress : PVOID;
	DestinationSize : UDINT;
END_VAR
END_METHOD

END_INTERFACE

// ---- mobject-collections/Interfaces/Collections/Nodes/I_LinkedListNode.TcIO
INTERFACE I_LinkedListNode EXTENDS I_CollectionNode

PROPERTY PUBLIC Next : I_LinkedListNode
GET
END_GET
SET
END_SET
END_PROPERTY

PROPERTY PUBLIC Previous : I_LinkedListNode
GET
END_GET
SET
END_SET
END_PROPERTY

END_INTERFACE

// ---- mobject-collections/Interfaces/Collections/Nodes/I_ListNode.TcIO
INTERFACE I_ListNode EXTENDS I_CollectionNode;

END_INTERFACE

// ---- mobject-collections/Interfaces/KeyValueCollections/Events/I_KeyValueCollectionChangedEvent.TcIO
INTERFACE I_KeyValueCollectionChangedEvent EXTENDS I_Event

PROPERTY PUBLIC Target : I_KeyValueCollection
GET
END_GET
END_PROPERTY

END_INTERFACE

// ---- mobject-collections/Interfaces/KeyValueCollections/Events/I_KeyValueCollectionDisposedEvent.TcIO
INTERFACE I_KeyValueCollectionDisposedEvent EXTENDS I_Event

PROPERTY PUBLIC Target : I_KeyValueCollection
GET
END_GET
END_PROPERTY

END_INTERFACE

// ---- mobject-collections/Interfaces/KeyValueCollections/I_Dictionary.TcIO
INTERFACE I_Dictionary EXTENDS I_KeyValueCollection

METHOD PUBLIC AddOrUpdate
VAR_INPUT
	Key : T_MAXSTRING;
	Value : ANY;
END_VAR
END_METHOD

METHOD PUBLIC Clear
VAR_INPUT
END_VAR
END_METHOD

METHOD PUBLIC ContainsKey : BOOL
VAR_INPUT
	Key : T_MAXSTRING;
END_VAR
END_METHOD

METHOD PUBLIC GetKeys : I_Collection
END_METHOD

PROPERTY IsEmpty : BOOL
GET
END_GET
END_PROPERTY

METHOD PUBLIC Remove
VAR_INPUT
	Key : T_MAXSTRING;
END_VAR
END_METHOD

METHOD PUBLIC TryAdd : BOOL
VAR_INPUT
	Key : T_MAXSTRING;
	Value : ANY;
END_VAR
END_METHOD

METHOD PUBLIC TryGetValue : BOOL
VAR_INPUT
	Key : T_MAXSTRING;
	Destination	: ANY;
END_VAR
END_METHOD

METHOD PUBLIC TryGetValueTo : BOOL
VAR_INPUT
	Key : T_MAXSTRING;
	DestinationAddress : PVOID;
	DestinationSize : UDINT;
END_VAR
END_METHOD

END_INTERFACE

// ---- mobject-collections/Interfaces/KeyValueCollections/I_KeyValueCollection.TcIO
INTERFACE I_KeyValueCollection EXTENDS I_KeyValueEnumerable, I_Enumerable, I_Disposable, I_EventEmitter

END_INTERFACE

// ---- mobject-commands/_Internal/AsyncCommandStateMachine/I_AsyncCommandStateControl.TcIO
INTERFACE I_AsyncCommandStateControl

METHOD PUBLIC Error
VAR_INPUT
	ErrorId : UDINT;
END_VAR
END_METHOD

METHOD PUBLIC Next
VAR_INPUT
END_VAR
END_METHOD

END_INTERFACE

// ---- mobject-datatypes/Datatypes/Events/I_DatatypeAddedEvent.TcIO
INTERFACE I_DatatypeAddedEvent EXTENDS I_Event

PROPERTY PUBLIC Target : I_Datatype
GET
END_GET
END_PROPERTY

END_INTERFACE

// ---- mobject-datatypes/Datatypes/Events/I_EnumDatatypeAddedEvent.TcIO
INTERFACE I_EnumDatatypeAddedEvent EXTENDS I_Event

PROPERTY PUBLIC Target : I_EnumDatatype
GET
END_GET
END_PROPERTY

END_INTERFACE

// ---- mobject-datatypes/Datatypes/Interface/I_Datatypes.TcIO
INTERFACE I_Datatypes EXTENDS I_EventEmitter

METHOD PUBLIC Accept
VAR_INPUT
	Visitor : I_DatatypeVisitor;
END_VAR
END_METHOD

METHOD RegisterDatatype
VAR_INPUT
	Datatype : I_Datatype;
END_VAR
END_METHOD

METHOD PUBLIC SerializeTypeWith
VAR_INPUT
	Serializer : I_Serializer;
END_VAR
END_METHOD

METHOD PUBLIC TryGetAliasByIdentifier : BOOL
VAR_INPUT
	Identifier : T_MAXSTRING;
	Destination : REFERENCE TO I_AliasDatatype;
END_VAR
END_METHOD

METHOD PUBLIC TryGetArrayByIdentifier : BOOL
VAR_INPUT
	Identifier : T_MAXSTRING;
	Destination : REFERENCE TO I_ArrayDatatype;
END_VAR
END_METHOD

METHOD PUBLIC TryGetEnumByIdentifier : BOOL
VAR_INPUT
	Identifier : T_MAXSTRING;
	Destination : REFERENCE TO I_EnumDatatype;
END_VAR
END_METHOD

METHOD PUBLIC TryGetInterfaceByIdentifier : BOOL
VAR_INPUT
	Identifier : T_MAXSTRING;
	Destination : REFERENCE TO I_InterfaceDatatype;
END_VAR
END_METHOD

METHOD PUBLIC TryGetPrimitiveByTypeName : BOOL
VAR_INPUT
	TypeName : T_MAXSTRING;
	Destination : REFERENCE TO I_AliasDatatype;
END_VAR
END_METHOD

METHOD PUBLIC TryGetStructureByIdentifier : BOOL
VAR_INPUT
	Identifier : T_MAXSTRING;
	Destination : REFERENCE TO I_StructuredDatatype;
END_VAR
END_METHOD

END_INTERFACE

// ---- mobject-datatypes/DatatypeVisitor/I_DatatypeVisitor.TcIO
INTERFACE I_DatatypeVisitor

METHOD VisitDatatype
VAR_INPUT
	VisitingDatatype : I_Datatype;
END_VAR
END_METHOD

END_INTERFACE

// ---- mobject-datatypes/Primitive/Interfaces/I_BIT.TcIO
INTERFACE I_BIT EXTENDS I_Datatype

PROPERTY PUBLIC BitOffset : DWORD
GET
END_GET
END_PROPERTY

PROPERTY PUBLIC ByteOffset : PVOID
GET
END_GET
END_PROPERTY

PROPERTY PUBLIC Parent : I_StructuredDatatype
GET
END_GET
END_PROPERTY

PROPERTY PUBLIC Value : BOOL
GET
END_GET
SET
END_SET
END_PROPERTY

END_INTERFACE

// ---- mobject-datatypes/Primitive/Interfaces/I_BYTE.TcIO
INTERFACE I_BYTE EXTENDS I_Datatype

{warning disable C5410}
PROPERTY PUBLIC Value : REFERENCE TO BYTE
{warning restore C5410}
GET
END_GET
END_PROPERTY

END_INTERFACE

// ---- mobject-datatypes/Primitive/Interfaces/I_ANY.TcIO
INTERFACE I_ANY EXTENDS I_Datatype

METHOD PUBLIC CanBecome : BOOL
VAR_INPUT
	Target : I_Datatype;
END_VAR
END_METHOD

METHOD PUBLIC Clear
VAR_INPUT
END_VAR
END_METHOD

PROPERTY PUBLIC IsResolved : BOOL
GET
END_GET
END_PROPERTY

METHOD PUBLIC TryBecome : BOOL
VAR_INPUT
	Target : I_Datatype;
END_VAR
END_METHOD

END_INTERFACE

// ---- mobject-datatypes/Primitive/Interfaces/I_DINT.TcIO
INTERFACE I_DINT EXTENDS I_Datatype

{warning disable C5410}
PROPERTY PUBLIC Value : REFERENCE TO DINT
{warning restore C5410}
GET
END_GET
END_PROPERTY

END_INTERFACE

// ---- mobject-datatypes/Primitive/Interfaces/I_DT.TcIO
INTERFACE I_DT EXTENDS I_Datatype

{warning disable C5410}
PROPERTY PUBLIC Value : REFERENCE TO DT
{warning restore C5410}
GET
END_GET
END_PROPERTY

END_INTERFACE

// ---- mobject-datatypes/Primitive/Interfaces/I_DWORD.TcIO
INTERFACE I_DWORD EXTENDS I_Datatype

{warning disable C5410}
PROPERTY PUBLIC Value : REFERENCE TO DWORD
{warning restore C5410}
GET
END_GET
END_PROPERTY

END_INTERFACE

// ---- mobject-datatypes/Primitive/Interfaces/I_INT.TcIO
INTERFACE I_INT EXTENDS I_Datatype

{warning disable C5410}
PROPERTY PUBLIC Value : REFERENCE TO INT
{warning restore C5410}
GET
END_GET
END_PROPERTY

END_INTERFACE

// ---- mobject-datatypes/Primitive/Interfaces/I_LINT.TcIO
INTERFACE I_LINT EXTENDS I_Datatype

{warning disable C5410}
PROPERTY PUBLIC Value : REFERENCE TO LINT
{warning restore C5410}
GET
END_GET
END_PROPERTY

END_INTERFACE

// ---- mobject-datatypes/Primitive/Interfaces/I_LREAL.TcIO
INTERFACE I_LREAL EXTENDS I_Datatype

{warning disable C5410}
PROPERTY PUBLIC Value : REFERENCE TO LREAL
{warning restore C5410}
GET
END_GET
END_PROPERTY

END_INTERFACE

// ---- mobject-datatypes/Primitive/Interfaces/I_LWORD.TcIO
INTERFACE I_LWORD EXTENDS I_Datatype

{warning disable C5410}
PROPERTY PUBLIC Value : REFERENCE TO LWORD
{warning restore C5410}
GET
END_GET
END_PROPERTY

END_INTERFACE

// ---- mobject-datatypes/Primitive/Interfaces/I_PVOID.TcIO
INTERFACE I_PVOID EXTENDS I_Datatype

{warning disable C5410}
PROPERTY PUBLIC Value : REFERENCE TO PVOID
{warning restore C5410}
GET
END_GET
END_PROPERTY

END_INTERFACE

// ---- mobject-datatypes/Primitive/Interfaces/I_REAL.TcIO
INTERFACE I_REAL EXTENDS I_Datatype

{warning disable C5410}
PROPERTY PUBLIC Value : REFERENCE TO REAL
{warning restore C5410}
GET
END_GET
END_PROPERTY

END_INTERFACE

// ---- mobject-datatypes/Primitive/Interfaces/I_REFERENCE_TO.TcIO
INTERFACE I_REFERENCE_TO EXTENDS I_Datatype

PROPERTY PUBLIC IsValidReference : BOOL
GET
END_GET
END_PROPERTY

END_INTERFACE

// ---- mobject-datatypes/Primitive/Interfaces/I_SINT.TcIO
INTERFACE I_SINT EXTENDS I_Datatype

{warning disable C5410}
PROPERTY PUBLIC Value : REFERENCE TO SINT
{warning restore C5410}
GET
END_GET
END_PROPERTY

END_INTERFACE

// ---- mobject-datatypes/Primitive/Interfaces/I_TOD.TcIO
INTERFACE I_TOD EXTENDS I_Datatype

{warning disable C5410}
PROPERTY PUBLIC Value : REFERENCE TO TOD
{warning restore C5410}
GET
END_GET
END_PROPERTY

END_INTERFACE

// ---- mobject-datatypes/Primitive/Interfaces/I_TIME_OF_DAY.TcIO
INTERFACE I_TIME_OF_DAY EXTENDS I_Datatype

{warning disable C5410}
PROPERTY PUBLIC Value : REFERENCE TO TIME_OF_DAY
{warning restore C5410}
GET
END_GET
END_PROPERTY

END_INTERFACE

// ---- mobject-datatypes/Primitive/Interfaces/I_STRING.TcIO
INTERFACE I_STRING EXTENDS I_Datatype

{warning disable C5410}
PROPERTY PUBLIC Value : REFERENCE TO T_MaxString
{warning restore C5410}
GET
END_GET
END_PROPERTY

END_INTERFACE

// ---- mobject-datatypes/Primitive/Interfaces/I_BOOL.TcIO
INTERFACE I_BOOL EXTENDS I_Datatype

{warning disable C5410}
PROPERTY PUBLIC Value : REFERENCE TO BOOL
{warning restore C5410}
GET
END_GET
END_PROPERTY

END_INTERFACE

// ---- mobject-datatypes/Primitive/Interfaces/I_UDINT.TcIO
INTERFACE I_UDINT EXTENDS I_Datatype

{warning disable C5410}
PROPERTY PUBLIC Value : REFERENCE TO UDINT
{warning restore C5410}
GET
END_GET
END_PROPERTY

END_INTERFACE

// ---- mobject-datatypes/Primitive/Interfaces/I_UINT.TcIO
INTERFACE I_UINT EXTENDS I_Datatype

{warning disable C5410}
PROPERTY PUBLIC Value : REFERENCE TO UINT
{warning restore C5410}
GET
END_GET
END_PROPERTY

END_INTERFACE

// ---- mobject-datatypes/Primitive/Interfaces/I_ULINT.TcIO
INTERFACE I_ULINT EXTENDS I_Datatype

{warning disable C5410}
PROPERTY PUBLIC Value : REFERENCE TO ULINT
{warning restore C5410}
GET
END_GET
END_PROPERTY

END_INTERFACE

// ---- mobject-datatypes/Primitive/Interfaces/I_USINT.TcIO
INTERFACE I_USINT EXTENDS I_Datatype

{warning disable C5410}
PROPERTY PUBLIC Value : REFERENCE TO USINT
{warning restore C5410}
GET
END_GET
END_PROPERTY

END_INTERFACE

// ---- mobject-datatypes/Primitive/Interfaces/I_WORD.TcIO
INTERFACE I_WORD EXTENDS I_Datatype

{warning disable C5410}
PROPERTY PUBLIC Value : REFERENCE TO WORD
{warning restore C5410}
GET
END_GET
END_PROPERTY

END_INTERFACE

// ---- mobject-datatypes/_Internal/Datatype/Interface/I_AliasDatatype.TcIO
INTERFACE I_AliasDatatype EXTENDS I_UserDefinedDatatype

PROPERTY PUBLIC BaseDatatype : I_Datatype
GET
END_GET
END_PROPERTY

END_INTERFACE

// ---- mobject-datatypes/_Internal/Datatype/Interface/I_ArrayDatatype_1D.TcIO
INTERFACE I_ArrayDatatype_1D EXTENDS I_ArrayDatatype

METHOD PUBLIC TryGetElementAsDatatypeByIndex : BOOL
VAR_INPUT
	Index : DINT;
	Destination : REFERENCE TO I_Datatype;
END_VAR
END_METHOD

END_INTERFACE

// ---- mobject-datatypes/_Internal/Datatype/Interface/I_ArrayDatatype_3D.TcIO
INTERFACE I_ArrayDatatype_3D EXTENDS I_ArrayDatatype

METHOD PUBLIC TryGetElementAsDatatypeByIndex : BOOL
VAR_INPUT
	Index1 : DINT;
	Index2 : DINT;
	Index3 : DINT;
	Destination : REFERENCE TO I_Datatype;
END_VAR
END_METHOD

END_INTERFACE

// ---- mobject-datatypes/_Internal/Datatype/Interface/I_Datatype.TcIO
INTERFACE I_Datatype extends I_Serializable, I_Deserializable, I_Disposable

METHOD PUBLIC Accept
VAR_INPUT
	Visitor : I_DatatypeVisitor;
END_VAR
END_METHOD

PROPERTY PUBLIC Address : PVOID
GET
END_GET
END_PROPERTY

METHOD PUBLIC ClearReference
VAR_INPUT
END_VAR
END_METHOD

METHOD Clone : I_Datatype
END_METHOD

METHOD PUBLIC IsEquivalentTo : BOOL
VAR_INPUT
	Datatype : I_Datatype;
END_VAR
END_METHOD

PROPERTY PUBLIC IsNull : BOOL
GET
END_GET
END_PROPERTY

PROPERTY PUBLIC IsUserDefined : BOOL
GET
END_GET
END_PROPERTY

PROPERTY PUBLIC Root : I_Datatype
GET
END_GET
END_PROPERTY

METHOD PUBLIC SerializeTypeWith
VAR_INPUT
	Serializer : I_Serializer;
END_VAR
END_METHOD

PROPERTY PUBLIC Size : UDINT
GET
END_GET
END_PROPERTY

METHOD PUBLIC TryConvertTo : BOOL
VAR_INPUT
	Destination : ANY;
END_VAR
END_METHOD

METHOD PUBLIC TryConvertTo_ : BOOL
VAR_INPUT
	Destination : I_Datatype;
END_VAR
END_METHOD

METHOD PUBLIC TryCopyFrom : BOOL
VAR_INPUT
	Source : I_Datatype;
END_VAR
END_METHOD

METHOD PUBLIC ABSTRACT TryDeserializeFrom : BOOL
VAR_INPUT
	Deserializer : I_Deserializer;
	Feedback : I_DeserializerFeedback;
END_VAR
END_METHOD

METHOD TryMakeReferenceTo : BOOL
VAR_INPUT
	Target : I_Datatype;
END_VAR
END_METHOD

METHOD PUBLIC TryResolveAs_ANY : BOOL
VAR_INPUT
	Destination : REFERENCE TO I_ANY;
END_VAR
END_METHOD

METHOD PUBLIC TryResolveAs_BIT : BOOL
VAR_INPUT
	Destination : REFERENCE TO I_BIT;
END_VAR
END_METHOD

METHOD PUBLIC TryResolveAs_BOOL : BOOL
VAR_INPUT
	Destination : REFERENCE TO I_BOOL;
END_VAR
END_METHOD

METHOD PUBLIC TryResolveAs_BYTE : BOOL
VAR_INPUT
	Destination : REFERENCE TO I_BYTE;
END_VAR
END_METHOD

METHOD PUBLIC TryResolveAs_DINT : BOOL
VAR_INPUT
	Destination : REFERENCE TO I_DINT;
END_VAR
END_METHOD

METHOD PUBLIC TryResolveAs_DT : BOOL
VAR_INPUT
	Destination : REFERENCE TO I_DT;
END_VAR
END_METHOD

METHOD PUBLIC TryResolveAs_DWORD : BOOL
VAR_INPUT
	Destination : REFERENCE TO I_DWORD;
END_VAR
END_METHOD

METHOD PUBLIC TryResolveAs_INT : BOOL
VAR_INPUT
	Destination : REFERENCE TO I_INT;
END_VAR
END_METHOD

METHOD PUBLIC TryResolveAs_LINT : BOOL
VAR_INPUT
	Destination : REFERENCE TO I_LINT;
END_VAR
END_METHOD

METHOD PUBLIC TryResolveAs_LREAL : BOOL
VAR_INPUT
	Destination : REFERENCE TO I_LREAL;
END_VAR
END_METHOD

METHOD PUBLIC TryResolveAs_LWORD : BOOL
VAR_INPUT
	Destination : REFERENCE TO I_LWORD;
END_VAR
END_METHOD

METHOD PUBLIC TryResolveAs_PVOID : BOOL
VAR_INPUT
	Destination : REFERENCE TO I_PVOID;
END_VAR
END_METHOD

METHOD PUBLIC TryResolveAs_REAL : BOOL
VAR_INPUT
	Destination : REFERENCE TO I_REAL;
END_VAR
END_METHOD

METHOD PUBLIC TryResolveAs_REFERENCE_TO : BOOL
VAR_INPUT
	Destination : REFERENCE TO I_REFERENCE_TO;
END_VAR
END_METHOD

METHOD PUBLIC TryResolveAs_SINT : BOOL
VAR_INPUT
	Destination : REFERENCE TO I_SINT;
END_VAR
END_METHOD

METHOD PUBLIC TryResolveAs_STRING : BOOL
VAR_INPUT
	Destination : REFERENCE TO I_STRING;
END_VAR
END_METHOD

METHOD PUBLIC TryResolveAs_TIME_OF_DAY : BOOL
VAR_INPUT
	Destination : REFERENCE TO I_TIME_OF_DAY;
END_VAR
END_METHOD

METHOD PUBLIC TryResolveAs_TOD : BOOL
VAR_INPUT
	Destination : REFERENCE TO I_TOD;
END_VAR
END_METHOD

METHOD PUBLIC TryResolveAs_UDINT : BOOL
VAR_INPUT
	Destination : REFERENCE TO I_UDINT;
END_VAR
END_METHOD

METHOD PUBLIC TryResolveAs_UINT : BOOL
VAR_INPUT
	Destination : REFERENCE TO I_UINT;
END_VAR
END_METHOD

METHOD PUBLIC TryResolveAs_ULINT : BOOL
VAR_INPUT
	Destination : REFERENCE TO I_ULINT;
END_VAR
END_METHOD

METHOD PUBLIC TryResolveAs_USINT : BOOL
VAR_INPUT
	Destination : REFERENCE TO I_USINT;
END_VAR
END_METHOD

METHOD PUBLIC TryResolveAs_WORD : BOOL
VAR_INPUT
	Destination : REFERENCE TO I_WORD;
END_VAR
END_METHOD

METHOD PUBLIC TryResolveAsAliasDatatype : BOOL
VAR_INPUT
	Destination : REFERENCE TO I_AliasDatatype;
END_VAR
END_METHOD

METHOD PUBLIC TryResolveAsArrayDatatype : BOOL
VAR_INPUT
	Destination : REFERENCE TO I_ArrayDatatype;
END_VAR
END_METHOD

METHOD PUBLIC TryResolveAsBitDatatype : BOOL
VAR_INPUT
	Destination : REFERENCE TO I_BIT;
END_VAR
END_METHOD

METHOD PUBLIC TryResolveAsEnumDatatype : BOOL
VAR_INPUT
	Destination : REFERENCE TO I_EnumDatatype;
END_VAR
END_METHOD

METHOD PUBLIC TryResolveAsInterfaceDatatype : BOOL
VAR_INPUT
	Destination : REFERENCE TO I_InterfaceDatatype;
END_VAR
END_METHOD

METHOD PUBLIC TryResolveAsStructuredDatatype : BOOL
VAR_INPUT
	Destination : REFERENCE TO I_StructuredDatatype;
END_VAR
END_METHOD

METHOD PUBLIC TryResolveAsUserDefinedDatatype : BOOL
VAR_INPUT
	Destination : REFERENCE TO I_UserDefinedDatatype;
END_VAR
END_METHOD

PROPERTY PUBLIC TypeName : T_MAXSTRING
GET
END_GET
END_PROPERTY

END_INTERFACE

// ---- mobject-datatypes/_Internal/Datatype/Interface/I_EnumDatatype.TcIO
INTERFACE I_EnumDatatype EXTENDS I_UserDefinedDatatype

END_INTERFACE

// ---- mobject-datatypes/_Internal/Datatype/Interface/I_InterfaceDatatype.TcIO
INTERFACE I_InterfaceDatatype EXTENDS I_Datatype

PROPERTY PUBLIC Identifier : T_MAXSTRING
GET
END_GET
END_PROPERTY

METHOD PUBLIC TryCopyContentFrom : BOOL
VAR_INPUT
	Source : I_InterfaceDatatype;
END_VAR
END_METHOD

END_INTERFACE

// ---- mobject-datatypes/_Internal/Datatype/Interface/I_StructuredDatatype.TcIO
INTERFACE I_StructuredDatatype EXTENDS I_UserDefinedDatatype, I_HostStructureMembers

END_INTERFACE

// ---- mobject-datatypes/_Internal/Datatype/Interface/I_ArrayDatatype.TcIO
INTERFACE I_ArrayDatatype EXTENDS I_UserDefinedDatatype

PROPERTY Dimention : UDINT
GET
END_GET
END_PROPERTY

METHOD TryGetLowerBound : BOOL
VAR_INPUT
	Dimention : UDINT;
	Destination : REFERENCE TO DINT;
END_VAR
END_METHOD

METHOD TryGetUpperBound : BOOL
VAR_INPUT
	Dimention : UDINT;
	Destination : REFERENCE TO DINT;
END_VAR
END_METHOD

METHOD PUBLIC TryResolveAs1DArrayDatatype : BOOL
VAR_INPUT
	Destination : REFERENCE TO I_ArrayDatatype_1D;
END_VAR
END_METHOD

METHOD PUBLIC TryResolveAs2DArrayDatatype : BOOL
VAR_INPUT
	Destination : REFERENCE TO I_ArrayDatatype_2D;
END_VAR
END_METHOD

METHOD PUBLIC TryResolveAs3DArrayDatatype : BOOL
VAR_INPUT
	Destination : REFERENCE TO I_ArrayDatatype_3D;
END_VAR
END_METHOD

END_INTERFACE

// ---- mobject-datatypes/_Internal/Datatype/Interface/I_UserDefinedDatatype.TcIO
INTERFACE I_UserDefinedDatatype EXTENDS I_Datatype

PROPERTY PUBLIC Identifier : T_MAXSTRING
GET
END_GET
END_PROPERTY

END_INTERFACE

// ---- mobject-datatypes/_Internal/StructureMembers/Interface/I_HostStructureMembers.TcIO
INTERFACE I_HostStructureMembers EXTENDS __SYSTEM.IQueryInterface

PROPERTY PUBLIC Members : I_StructureMembers
GET
END_GET
END_PROPERTY

END_INTERFACE

// ---- mobject-deserialization/Interfaces/I_Deserializer.TcIO
INTERFACE I_Deserializer EXTENDS I_Disposable

METHOD PUBLIC Clone : I_Deserializer
END_METHOD

METHOD GetArray : I_Deserializer
VAR_INPUT
END_VAR
END_METHOD

METHOD GetArrayEnumerator : I_DeserializerArrayForwardEnumerator
VAR_INPUT
END_VAR
END_METHOD

METHOD GetElementByIndex : I_Deserializer
VAR_INPUT
	Index : UDINT;
END_VAR
END_METHOD

METHOD GetKeyArray : I_Deserializer
VAR_INPUT
	Key : T_MAXSTRING;
END_VAR
END_METHOD

METHOD GetKeyObject : I_Deserializer
VAR_INPUT
	Key : T_MAXSTRING;
END_VAR
END_METHOD

METHOD GetObject : I_Deserializer
VAR_INPUT
END_VAR
END_METHOD

METHOD GetObjectEnumerator : I_DeserializerObjectForwardEnumerator
VAR_INPUT
END_VAR
END_METHOD

METHOD TryDeserializeKeyToObject : BOOL
VAR_INPUT
	Key : T_MAXSTRING;
	Object : I_Deserializable;
	Feedback : I_DeserializerFeedback;
END_VAR
END_METHOD

METHOD TryDeserializeToObject : BOOL
VAR_INPUT
	Object : I_Deserializable;
	Feedback : I_DeserializerFeedback;
END_VAR
END_METHOD

METHOD TryGetBase64 : BOOL
VAR_INPUT
	pBytes : POINTER TO BYTE;
	nBytes : DINT;
	Feedback : I_DeserializerFeedback;
END_VAR
END_METHOD

METHOD TryGetBool : BOOL
VAR_INPUT
	Destination : REFERENCE TO BOOL;
	Feedback : I_DeserializerFeedback;
END_VAR
END_METHOD

METHOD TryGetByte : BOOL
VAR_INPUT
	Destination : REFERENCE TO BYTE;
	Feedback : I_DeserializerFeedback;
END_VAR
END_METHOD

METHOD TryGetDateTime : BOOL
VAR_INPUT
	Destination : REFERENCE TO DATE_AND_TIME;
	Feedback : I_DeserializerFeedback;
END_VAR
END_METHOD

METHOD TryGetDcTime : BOOL
VAR_INPUT
	Destination : REFERENCE TO DCTIME;
	Feedback : I_DeserializerFeedback;
END_VAR
END_METHOD

METHOD TryGetDint : BOOL
VAR_INPUT
	Destination : REFERENCE TO DINT;
	Feedback : I_DeserializerFeedback;
END_VAR
END_METHOD

METHOD TryGetDword : BOOL
VAR_INPUT
	Destination : REFERENCE TO DWORD;
	Feedback : I_DeserializerFeedback;
END_VAR
END_METHOD

METHOD TryGetElementByIndex : BOOL
VAR_INPUT
	Index : UDINT;
	Destination : REFERENCE TO I_Deserializer;
	Feedback : I_DeserializerFeedback;
END_VAR
END_METHOD

METHOD TryGetFileTime : BOOL
VAR_INPUT
	Destination : REFERENCE TO FILETIME;
	Feedback : I_DeserializerFeedback;
END_VAR
END_METHOD

METHOD TryGetHexAsBytes : BOOL
VAR_INPUT
	pBytes : POINTER TO BYTE;
	nBytes : DINT;
	Feedback : I_DeserializerFeedback;
END_VAR
END_METHOD

METHOD TryGetInt : BOOL
VAR_INPUT
	Destination : REFERENCE TO INT;
	Feedback : I_DeserializerFeedback;
END_VAR
END_METHOD

METHOD TryGetKeyBase64 : BOOL
VAR_INPUT
	Key : T_MAXSTRING;
	pBytes : POINTER TO BYTE;
	nBytes : DINT;
	Feedback : I_DeserializerFeedback;
END_VAR
END_METHOD

METHOD TryGetKeyBool : BOOL
VAR_INPUT
	Key : T_MAXSTRING;
	Destination : REFERENCE TO BOOL;
	Feedback : I_DeserializerFeedback;
END_VAR
END_METHOD

METHOD TryGetKeyByte : BOOL
VAR_INPUT
	Key : T_MAXSTRING;
	Destination : REFERENCE TO BYTE;
	Feedback : I_DeserializerFeedback;
END_VAR
END_METHOD

METHOD TryGetKeyDateTime : BOOL
VAR_INPUT
	Key : T_MAXSTRING;
	Destination : REFERENCE TO DATE_AND_TIME;
	Feedback : I_DeserializerFeedback;
END_VAR
END_METHOD

METHOD TryGetKeyDcTime : BOOL
VAR_INPUT
	Key : T_MAXSTRING;
	Destination : REFERENCE TO DCTIME;
	Feedback : I_DeserializerFeedback;
END_VAR
END_METHOD

METHOD TryGetKeyDint : BOOL
VAR_INPUT
	Key : T_MAXSTRING;
	Destination : REFERENCE TO DINT;
	Feedback : I_DeserializerFeedback;
END_VAR
END_METHOD

METHOD TryGetKeyDword : BOOL
VAR_INPUT
	Key : T_MAXSTRING;
	Destination : REFERENCE TO DWORD;
	Feedback : I_DeserializerFeedback;
END_VAR
END_METHOD

METHOD TryGetKeyFileTime : BOOL
VAR_INPUT
	Key : T_MAXSTRING;
	Destination : REFERENCE TO FILETIME;
	Feedback : I_DeserializerFeedback;
END_VAR
END_METHOD

METHOD TryGetKeyHexAsBytes : BOOL
VAR_INPUT
	Key : T_MAXSTRING;
	pBytes : POINTER TO BYTE;
	nBytes : DINT;
	Feedback : I_DeserializerFeedback;
END_VAR
END_METHOD

METHOD TryGetKeyInt : BOOL
VAR_INPUT
	Key : T_MAXSTRING;
	Destination : REFERENCE TO INT;
	Feedback : I_DeserializerFeedback;
END_VAR
END_METHOD

METHOD TryGetKeyLint : BOOL
VAR_INPUT
	Key : T_MAXSTRING;
	Destination : REFERENCE TO LINT;
	Feedback : I_DeserializerFeedback;
END_VAR
END_METHOD

METHOD TryGetKeyLreal : BOOL
VAR_INPUT
	Key : T_MAXSTRING;
	Destination : REFERENCE TO LREAL;
	Feedback : I_DeserializerFeedback;
END_VAR
END_METHOD

METHOD TryGetKeyLtime : BOOL
VAR_INPUT
	Key : T_MAXSTRING;
	Destination : REFERENCE TO LTIME;
	Feedback : I_DeserializerFeedback;
END_VAR
END_METHOD

METHOD TryGetKeyLword : BOOL
VAR_INPUT
	Key : T_MAXSTRING;
	Destination : REFERENCE TO LWORD;
	Feedback : I_DeserializerFeedback;
END_VAR
END_METHOD

METHOD TryGetKeyReal : BOOL
VAR_INPUT
	Key : T_MAXSTRING;
	Destination : REFERENCE TO REAL;
	Feedback : I_DeserializerFeedback;
END_VAR
END_METHOD

METHOD TryGetKeySint : BOOL
VAR_INPUT
	Key : T_MAXSTRING;
	Destination : REFERENCE TO SINT;
	Feedback : I_DeserializerFeedback;
END_VAR
END_METHOD

METHOD TryGetKeyString : BOOL
VAR_INPUT
	Key : T_MAXSTRING;
	Destination : REFERENCE TO T_MAXSTRING;
	Feedback : I_DeserializerFeedback;
END_VAR
END_METHOD

METHOD TryGetKeyStringEx : BOOL
VAR_INPUT
	Key : T_MAXSTRING;
	DestinationAddress : POINTER TO STRING;
	DestinationSize : UDINT;
	Feedback : I_DeserializerFeedback;
END_VAR
END_METHOD

METHOD TryGetKeyTime : BOOL
VAR_INPUT
	Key : T_MAXSTRING;
	Destination : REFERENCE TO TIME;
	Feedback : I_DeserializerFeedback;
END_VAR
END_METHOD

METHOD TryGetKeyTod : BOOL
VAR_INPUT
	Key : T_MAXSTRING;
	Destination : REFERENCE TO TOD;
	Feedback : I_DeserializerFeedback;
END_VAR
END_METHOD

METHOD TryGetKeyUdint : BOOL
VAR_INPUT
	Key : T_MAXSTRING;
	Destination : REFERENCE TO UDINT;
	Feedback : I_DeserializerFeedback;
END_VAR
END_METHOD

METHOD TryGetKeyUint : BOOL
VAR_INPUT
	Key : T_MAXSTRING;
	Destination : REFERENCE TO UINT;
	Feedback : I_DeserializerFeedback;
END_VAR
END_METHOD

METHOD TryGetKeyUlint : BOOL
VAR_INPUT
	Key : T_MAXSTRING;
	Destination : REFERENCE TO ULINT;
	Feedback : I_DeserializerFeedback;
END_VAR
END_METHOD

METHOD TryGetKeyUsint : BOOL
VAR_INPUT
	Key : T_MAXSTRING;
	Destination : REFERENCE TO USINT;
	Feedback : I_DeserializerFeedback;
END_VAR
END_METHOD

METHOD TryGetKeyWord : BOOL
VAR_INPUT
	Key : T_MAXSTRING;
	Destination : REFERENCE TO WORD;
	Feedback : I_DeserializerFeedback;
END_VAR
END_METHOD

METHOD TryGetLint : BOOL
VAR_INPUT
	Destination : REFERENCE TO LINT;
	Feedback : I_DeserializerFeedback;
END_VAR
END_METHOD

METHOD TryGetLreal : BOOL
VAR_INPUT
	Destination : REFERENCE TO LREAL;
	Feedback : I_DeserializerFeedback;
END_VAR
END_METHOD

METHOD TryGetLtime : BOOL
VAR_INPUT
	Destination : REFERENCE TO LTIME;
	Feedback : I_DeserializerFeedback;
END_VAR
END_METHOD

METHOD TryGetLword : BOOL
VAR_INPUT
	Destination : REFERENCE TO LWORD;
	Feedback : I_DeserializerFeedback;
END_VAR
END_METHOD

METHOD TryGetReal : BOOL
VAR_INPUT
	Destination : REFERENCE TO REAL;
	Feedback : I_DeserializerFeedback;
END_VAR
END_METHOD

METHOD TryGetSint : BOOL
VAR_INPUT
	Destination : REFERENCE TO SINT;
	Feedback : I_DeserializerFeedback;
END_VAR
END_METHOD

METHOD TryGetString : BOOL
VAR_INPUT
	Destination : REFERENCE TO T_MAXSTRING;
	Feedback : I_DeserializerFeedback;
END_VAR
END_METHOD

METHOD TryGetStringEx : BOOL
VAR_INPUT
	DestinationAddress : POINTER TO STRING;
	DestinationSize : UDINT;
	Feedback : I_DeserializerFeedback;
END_VAR
END_METHOD

METHOD TryGetTime : BOOL
VAR_INPUT
	Destination : REFERENCE TO TIME;
	Feedback : I_DeserializerFeedback;
END_VAR
END_METHOD

METHOD TryGetTod : BOOL
VAR_INPUT
	Destination : REFERENCE TO TOD;
	Feedback : I_DeserializerFeedback;
END_VAR
END_METHOD

METHOD TryGetUdint : BOOL
VAR_INPUT
	Destination : REFERENCE TO UDINT;
	Feedback : I_DeserializerFeedback;
END_VAR
END_METHOD

METHOD TryGetUint : BOOL
VAR_INPUT
	Destination : REFERENCE TO UINT;
	Feedback : I_DeserializerFeedback;
END_VAR
END_METHOD

METHOD TryGetUlint : BOOL
VAR_INPUT
	Destination : REFERENCE TO ULINT;
	Feedback : I_DeserializerFeedback;
END_VAR
END_METHOD

METHOD TryGetUsint : BOOL
VAR_INPUT
	Destination : REFERENCE TO USINT;
	Feedback : I_DeserializerFeedback;
END_VAR
END_METHOD

METHOD TryGetWord : BOOL
VAR_INPUT
	Destination : REFERENCE TO WORD;
	Feedback : I_DeserializerFeedback;
END_VAR
END_METHOD

END_INTERFACE

// ---- mobject-deserialization/Interfaces/I_DeserializerArrayForwardEnumerator.TcIO
INTERFACE I_DeserializerArrayForwardEnumerator EXTENDS I_Disposable

PROPERTY PUBLIC Current : I_Deserializer
GET
END_GET
END_PROPERTY

PROPERTY Index : DINT
GET
END_GET
END_PROPERTY

PROPERTY IsValid : BOOL
GET
END_GET
END_PROPERTY

METHOD MoveNext : BOOL
VAR_INPUT
END_VAR
END_METHOD

END_INTERFACE

// ---- mobject-deserialization/Interfaces/I_DeserializerFeedback.TcIO
INTERFACE I_DeserializerFeedback

METHOD PUBLIC LogDeserializationFailedError
VAR_INPUT
	Message : T_MAXSTRING;
END_VAR
END_METHOD

METHOD PUBLIC LogError
VAR_INPUT
	Error : I_Error;
END_VAR
END_METHOD

METHOD PUBLIC LogIncorrectKeyTypeError
VAR_INPUT
	ExpectedType : T_MAXSTRING;
	ActualKey : T_MAXSTRING;
END_VAR
END_METHOD

METHOD PUBLIC LogIncorrectTypeError
VAR_INPUT
	ExpectedType : T_MAXSTRING;
END_VAR
END_METHOD

METHOD PUBLIC LogInvalidKeyError
VAR_INPUT
END_VAR
END_METHOD

METHOD PUBLIC LogMissingKeyError
VAR_INPUT
	ExpectedKey : T_MAXSTRING;
END_VAR
END_METHOD

END_INTERFACE

// ---- mobject-deserialization/Interfaces/I_DeserializerObjectForwardEnumerator.TcIO
INTERFACE I_DeserializerObjectForwardEnumerator EXTENDS I_Disposable

PROPERTY PUBLIC Current : I_Deserializer
GET
END_GET
END_PROPERTY

PROPERTY IsValid : BOOL
GET
END_GET
END_PROPERTY

PROPERTY Key : T_MAXSTRING
GET
END_GET
END_PROPERTY

METHOD MoveNext : BOOL
VAR_INPUT
END_VAR
END_METHOD

END_INTERFACE

// ---- mobject-errors/Interfaces/I_Error.TcIO
INTERFACE I_Error EXTENDS I_Serializable, I_Disposable

METHOD PUBLIC Accept
VAR_INPUT
	Visitor : I_ErrorVisitor;
END_VAR
END_METHOD

PROPERTY ErrorType : T_MAXSTRING
GET
END_GET
END_PROPERTY

METHOD PUBLIC IsSameAs : BOOL
VAR_INPUT
	Error : I_Error;
END_VAR
END_METHOD

PROPERTY Message : T_MAXSTRING
GET
END_GET
END_PROPERTY

END_INTERFACE

// ---- mobject-errors/Interfaces/I_ErrorVisitor.TcIO
INTERFACE I_ErrorVisitor

METHOD VisitError
VAR_INPUT
	VisitingError : I_Error;
END_VAR
END_METHOD

END_INTERFACE

// ---- mobject-events/Interfaces/I_Event.TcIO
INTERFACE I_Event EXTENDS __SYSTEM.IQueryInterface

END_INTERFACE

// ---- mobject-events/_Internal/EventHandlerItem/I_EventHandlerItem.TcIO
INTERFACE I_EventHandlerItem EXTENDS I_Disposable

METHOD PUBLIC Emit : BOOL
VAR_INPUT
	EventName : T_MaxString;
	Event : I_Event;
END_VAR
END_METHOD

METHOD PUBLIC EqualTo : BOOL
VAR_INPUT
	Name : T_MaxString;
	Handler : I_EventHandler;
END_VAR
END_METHOD

PROPERTY PUBLIC Next : I_EventHandlerItem
GET
END_GET
SET
END_SET
END_PROPERTY

PROPERTY PUBLIC Previous : I_EventHandlerItem
GET
END_GET
SET
END_SET
END_PROPERTY

END_INTERFACE

// ---- mobject-enumerable/Interfaces/Enumerators/I_ForwardEnumerator.TcIO
INTERFACE I_ForwardEnumerator EXTENDS I_Disposable

PROPERTY PUBLIC IsValid : BOOL
GET
END_GET
END_PROPERTY

METHOD PUBLIC MoveNext : BOOL
END_METHOD

METHOD PUBLIC Reset
END_METHOD

METHOD PUBLIC TryGet : BOOL;
VAR_INPUT
    Destination : ANY;
END_VAR
END_METHOD

METHOD PUBLIC TryGetTo : BOOL;
VAR_INPUT
    DestinationAddress : PVOID;
    DestinationSize : UDINT;
END_VAR
END_METHOD

END_INTERFACE

// ---- mobject-enumerable/Interfaces/I_Enumerable.TcIO
INTERFACE I_Enumerable EXTENDS __SYSTEM.IQueryInterface

METHOD PUBLIC GetEnumerator : I_ForwardEnumerator
END_METHOD

END_INTERFACE

// ---- mobject-enumerable/Interfaces/I_KeyValueEnumerable.TcIO
INTERFACE I_KeyValueEnumerable EXTENDS __SYSTEM.IQueryInterface

METHOD PUBLIC GetKeyValueEnumerator : I_KeyValueForwardEnumerator
END_METHOD

END_INTERFACE

// ---- mobject-json/JsonDeserializer/Events/I_JsonDeserializerDisposedEvent.TcIO
INTERFACE I_JsonDeserializerDisposedEvent EXTENDS I_Event

PROPERTY PUBLIC Target : I_JsonDeserializer
GET
END_GET
END_PROPERTY

END_INTERFACE

// ---- mobject-json/JsonDeserializer/I_JsonDeserializer.TcIO
INTERFACE I_JsonDeserializer EXTENDS I_Deserializer, I_EventEmitter, I_Disposable

END_INTERFACE

// ---- mobject-serialization/Interfaces/I_Serializable.TcIO
INTERFACE I_Serializable EXTENDS __SYSTEM.IQueryInterface

METHOD SerializeWith
VAR_INPUT
	Serializer : I_Serializer;
END_VAR
END_METHOD

END_INTERFACE

// ---- mobject-serialization/Interfaces/I_Serializer.TcIO
INTERFACE I_Serializer EXTENDS I_Disposable

METHOD PUBLIC AddBase64 : I_Serializer
VAR_INPUT
	pBytes : POINTER TO BYTE;
	nBytes : DINT;
END_VAR
END_METHOD

METHOD PUBLIC AddBool : I_Serializer
VAR_INPUT
	Value : BOOL;
END_VAR
END_METHOD

METHOD PUBLIC AddByte : I_Serializer
VAR_INPUT
	Value : BYTE;
END_VAR
END_METHOD

METHOD PUBLIC AddBytesAsHex : I_Serializer
VAR_INPUT
	pBytes : POINTER TO BYTE;
	nBytes : DINT;
END_VAR
END_METHOD

METHOD PUBLIC AddDateTime : I_Serializer
VAR_INPUT
	Value : DATE_AND_TIME;
END_VAR
END_METHOD

METHOD PUBLIC AddDcTime : I_Serializer
VAR_INPUT
	Value : DCTIME;
END_VAR
END_METHOD

METHOD PUBLIC AddDint : I_Serializer
VAR_INPUT
	Value : DINT;
END_VAR
END_METHOD

METHOD PUBLIC AddDword : I_Serializer
VAR_INPUT
	Value : DWORD;
END_VAR
END_METHOD

METHOD PUBLIC AddFileTime : I_Serializer
VAR_INPUT
	Value : FILETIME;
END_VAR
END_METHOD

METHOD PUBLIC AddInt : I_Serializer
VAR_INPUT
	Value : INT;
END_VAR
END_METHOD

METHOD PUBLIC AddKey : I_Serializer
VAR_INPUT
	Key : T_MAXSTRING;
END_VAR
END_METHOD

METHOD PUBLIC AddKeyBase64 : I_Serializer
VAR_INPUT
	Key : T_MAXSTRING;
	pBytes : POINTER TO BYTE;
	nBytes : DINT;
END_VAR
END_METHOD

METHOD PUBLIC AddKeyBool : I_Serializer
VAR_INPUT
	Key : T_MAXSTRING;
	Value : BOOL;
END_VAR
END_METHOD

METHOD PUBLIC AddKeyByte : I_Serializer
VAR_INPUT
	Key : T_MAXSTRING;
	Value : BYTE;
END_VAR
END_METHOD

METHOD PUBLIC AddKeyBytesAsHex : I_Serializer
VAR_INPUT
	Key : T_MAXSTRING;
	pBytes : POINTER TO BYTE;
	nBytes : DINT;
END_VAR
END_METHOD

METHOD PUBLIC AddKeyDateTime : I_Serializer
VAR_INPUT
	Key : T_MAXSTRING;
	Value : DATE_AND_TIME;
END_VAR
END_METHOD

METHOD PUBLIC AddKeyDcTime : I_Serializer
VAR_INPUT
	Key : T_MAXSTRING;
	Value : DCTIME;
END_VAR
END_METHOD

METHOD PUBLIC AddKeyDint : I_Serializer
VAR_INPUT
	Key : T_MAXSTRING;
	Value : DINT;
END_VAR
END_METHOD

METHOD PUBLIC AddKeyDword : I_Serializer
VAR_INPUT
	Key : T_MAXSTRING;
	Value : DWORD;
END_VAR
END_METHOD

METHOD PUBLIC AddKeyFileTime : I_Serializer
VAR_INPUT
	Key : T_MAXSTRING;
	Value : FILETIME;
END_VAR
END_METHOD

METHOD PUBLIC AddKeyInt : I_Serializer
VAR_INPUT
	Key : T_MAXSTRING;
	Value : INT;
END_VAR
END_METHOD

METHOD PUBLIC AddKeyLint : I_Serializer
VAR_INPUT
	Key : T_MAXSTRING;
	Value : LINT;
END_VAR
END_METHOD

METHOD PUBLIC AddKeyLreal : I_Serializer
VAR_INPUT
	Key : T_MAXSTRING;
	Value : LREAL;
END_VAR
END_METHOD

METHOD PUBLIC AddKeyLtime : I_Serializer
VAR_INPUT
	Key : T_MAXSTRING;
	Value : LTIME;
END_VAR
END_METHOD

METHOD PUBLIC AddKeyLword : I_Serializer
VAR_INPUT
	Key : T_MAXSTRING;
	Value : LWORD;
END_VAR
END_METHOD

METHOD PUBLIC AddKeyNull : I_Serializer
VAR_INPUT
	Key : T_MAXSTRING;
END_VAR
END_METHOD

METHOD PUBLIC AddKeyObject : I_Serializer
VAR_INPUT
	Key : T_MAXSTRING;
	Object : I_Serializable;
END_VAR
END_METHOD

METHOD PUBLIC AddKeyReal : I_Serializer
VAR_INPUT
	Key : T_MAXSTRING;
	Value : REAL;
END_VAR
END_METHOD

METHOD PUBLIC AddKeySint : I_Serializer
VAR_INPUT
	Key : T_MAXSTRING;
	Value : SINT;
END_VAR
END_METHOD

METHOD PUBLIC AddKeyString : I_Serializer
VAR_INPUT
	Key : T_MAXSTRING;
	Value : T_MAXSTRING;
END_VAR
END_METHOD

METHOD PUBLIC AddKeyStringByRef : I_Serializer
VAR_INPUT
	Key : T_MAXSTRING;
	Value : REFERENCE TO STRING;
END_VAR
END_METHOD

METHOD PUBLIC AddKeyTime : I_Serializer
VAR_INPUT
	Key : T_MAXSTRING;
	Value : TIME;
END_VAR
END_METHOD

METHOD PUBLIC AddKeyTod : I_Serializer
VAR_INPUT
	Key : T_MAXSTRING;
	Value : TOD;
END_VAR
END_METHOD

METHOD PUBLIC AddKeyUdint : I_Serializer
VAR_INPUT
	Key : T_MAXSTRING;
	Value : UDINT;
END_VAR
END_METHOD

METHOD PUBLIC AddKeyUint : I_Serializer
VAR_INPUT
	Key : T_MAXSTRING;
	Value : UINT;
END_VAR
END_METHOD

METHOD PUBLIC AddKeyUlint : I_Serializer
VAR_INPUT
	Key : T_MAXSTRING;
	Value : ULINT;
END_VAR
END_METHOD

METHOD PUBLIC AddKeyUsint : I_Serializer
VAR_INPUT
	Key : T_MAXSTRING;
	Value : USINT;
END_VAR
END_METHOD

METHOD PUBLIC AddKeyWord : I_Serializer
VAR_INPUT
	Key : T_MAXSTRING;
	Value : WORD;
END_VAR
END_METHOD

METHOD PUBLIC AddLint : I_Serializer
VAR_INPUT
	Value : LINT;
END_VAR
END_METHOD

METHOD PUBLIC AddLreal : I_Serializer
VAR_INPUT
	Value : LREAL;
END_VAR
END_METHOD

METHOD PUBLIC AddLtime : I_Serializer
VAR_INPUT
	Value : LTIME;
END_VAR
END_METHOD

METHOD PUBLIC AddLword : I_Serializer
VAR_INPUT
	Value : LWORD;
END_VAR
END_METHOD

METHOD PUBLIC AddNull : I_Serializer
VAR_INPUT
END_VAR
END_METHOD

METHOD PUBLIC AddObject
VAR_INPUT
	Object : I_Serializable;
END_VAR
END_METHOD

METHOD PUBLIC AddReal : I_Serializer
VAR_INPUT
	Value : REAL;
END_VAR
END_METHOD

METHOD PUBLIC AddSint : I_Serializer
VAR_INPUT
	Value : SINT;
END_VAR
END_METHOD

METHOD PUBLIC AddString : I_Serializer
VAR_INPUT
	Value : T_MAXSTRING;
END_VAR
END_METHOD

METHOD PUBLIC AddStringByRef : I_Serializer
VAR_INPUT
	Value : REFERENCE TO STRING;
END_VAR
END_METHOD

METHOD PUBLIC AddTime : I_Serializer
VAR_INPUT
	Value : TIME;
END_VAR
END_METHOD

METHOD PUBLIC AddTod : I_Serializer
VAR_INPUT
	Value : TOD;
END_VAR
END_METHOD

METHOD PUBLIC AddUdint : I_Serializer
VAR_INPUT
	Value : UDINT;
END_VAR
END_METHOD

METHOD PUBLIC AddUint : I_Serializer
VAR_INPUT
	Value : UINT;
END_VAR
END_METHOD

METHOD PUBLIC AddUlint : I_Serializer
VAR_INPUT
	Value : ULINT;
END_VAR
END_METHOD

METHOD PUBLIC AddUsint : I_Serializer
VAR_INPUT
	Value : USINT;
END_VAR
END_METHOD

METHOD PUBLIC AddWord : I_Serializer
VAR_INPUT
	Value : WORD;
END_VAR
END_METHOD

METHOD PUBLIC Clone : I_Serializer
END_METHOD

METHOD PUBLIC EndArray : I_Serializer
VAR_INPUT
END_VAR
END_METHOD

METHOD PUBLIC EndObject : I_Serializer
VAR_INPUT
END_VAR
END_METHOD

METHOD PUBLIC GetSerializedDataLength : UDINT
VAR_INPUT
END_VAR
END_METHOD

METHOD PUBLIC Reset
VAR_INPUT
END_VAR
END_METHOD

METHOD PUBLIC StartArray : I_Serializer
VAR_INPUT
END_VAR
END_METHOD

METHOD PUBLIC StartObject : I_Serializer
VAR_INPUT
END_VAR
END_METHOD

METHOD TryCopySerializedData : BOOL
VAR_INPUT
	DestinationAddress : PVOID;
	DestinationSize : UDINT;
END_VAR
END_METHOD

METHOD TryGetSerializedData : BOOL
VAR_INPUT
	DestinationAddress : PVOID;
	DestinationSize : UDINT;
END_VAR
END_METHOD

END_INTERFACE

// ---- mobject-server/RpcApi/I_RpcApi.TcIO
INTERFACE I_RpcApi

METHOD CyclicCall
VAR_INPUT
END_VAR
END_METHOD

METHOD RegisterAsynchronousRpcHandlersWith
VAR_INPUT
	Host : I_HostAsynchronousRpcHandlers;
END_VAR
END_METHOD

METHOD RegisterSynchronousRpcHandlersWith
VAR_INPUT
	Host : I_HostSynchronousRpcHandlers;
END_VAR
END_METHOD

END_INTERFACE

// ---- mobject-server/RpcHandler/I_AsynchronousRpcHandler.TcIO
INTERFACE I_AsynchronousRpcHandler EXTENDS __SYSTEM.IQueryInterface

METHOD Handle
VAR_INPUT
	Parameters : I_Deserializer;
	Response : I_AsynchronousRpcResponse;
END_VAR
END_METHOD

END_INTERFACE

// ---- mobject-server/RpcHandler/I_SynchronousRpcHandler.TcIO
INTERFACE I_SynchronousRpcHandler EXTENDS __SYSTEM.IQueryInterface

METHOD Handle
VAR_INPUT
	Parameters : I_Deserializer;
	Response : I_SynchronousRpcResponse;
END_VAR
END_METHOD

END_INTERFACE

// ---- mobject-server/RpcServer/I_RpcServer.TcIO
INTERFACE I_RpcServer

METHOD PUBLIC GetConfiguredHeaderSize : UDINT
VAR_INPUT
END_VAR
END_METHOD

METHOD PUBLIC GetConfiguredPayloadSize : UDINT
VAR_INPUT
END_VAR
END_METHOD

{attribute 'TcRpcEnable'}
METHOD PUBLIC HandleRequest : ResponseData;
VAR_INPUT
	SerializedHeader : STRING(ServerConfiguration.HEADER_STRING_SIZE);
	SerializedPayload : STRING(ServerConfiguration.PAYLOAD_STRING_SIZE);
END_VAR
END_METHOD

METHOD PUBLIC RegisterApi
VAR_INPUT
	RpcApi : I_RpcApi;
END_VAR
END_METHOD

METHOD PUBLIC RegisterAsynchronousRpcHandler
VAR_INPUT
	MethodName : T_MAXSTRING;
	Handler : I_AsynchronousRpcHandler;
END_VAR
END_METHOD

METHOD PUBLIC RegisterSynchronousRpcHandler
VAR_INPUT
	MethodName : T_MAXSTRING;
	Handler : I_SynchronousRpcHandler;
END_VAR
END_METHOD

END_INTERFACE

// ---- mobject-server/_Internal/AsyncResponse/HeaderAccessor/I_AsyncResponseHeaderAccessor.TcIO
INTERFACE I_AsyncResponseHeaderAccessor

METHOD PUBLIC TryGetResponseIdFromRequest : BOOL
VAR_INPUT
	Request : I_Request;
	Destination : ANY;
END_VAR
END_METHOD

METHOD PUBLIC TryGetSessionIdFromRequest : BOOL
VAR_INPUT
	Request : I_Request;
	Destination : REFERENCE TO T_MAXSTRING;
END_VAR
END_METHOD

METHOD PUBLIC TryGetSessionIdFromResponse : BOOL
VAR_INPUT
	Response : I_ServerResponse;
	Destination : ANY;
END_VAR
END_METHOD

END_INTERFACE

// ---- mobject-server/_Internal/AsyncResponse/Manager/I_AsyncResponseManager.TcIO
INTERFACE I_AsyncResponseManager

METHOD TryConvertResponseToAsyncResponseSessionData : BOOL
VAR_INPUT
	Response : I_ServerResponse;
	RetryDelayInMs : UDINT;
	Destination : REFERENCE TO I_AsyncResponseSessionData;
END_VAR
END_METHOD

METHOD PUBLIC TryHandleIncomingRequest : BOOL
VAR_INPUT
	Request : I_Request;
	Response : I_ServerResponse;
END_VAR
END_METHOD

END_INTERFACE

// ---- mobject-server/_Internal/AsyncResponse/SessionData/I_AsyncResponseSessionData.TcIO
INTERFACE I_AsyncResponseSessionData EXTENDS I_SessionData

METHOD PUBLIC Error
VAR_INPUT
	ErrorCode : T_MAXSTRING;
	Message : T_MAXSTRING;
END_VAR
END_METHOD

PROPERTY PUBLIC HasExpired : BOOL
GET
END_GET
END_PROPERTY

PROPERTY PUBLIC IsPending : BOOL
GET
END_GET
END_PROPERTY

METHOD PUBLIC Success
VAR_INPUT
END_VAR
END_METHOD

METHOD PUBLIC SuccessWithPayload
VAR_INPUT
	PayloadDataAddress : PVOID;
	PayloadDataSize : UDINT;
END_VAR
END_METHOD

PROPERTY PUBLIC SuggestedRetryDelayInMs : UDINT
GET
END_GET
SET
END_SET
END_PROPERTY

METHOD PUBLIC TryUpdateServerResponse : BOOL
VAR_INPUT
	Response : I_ServerResponse;
END_VAR
END_METHOD

END_INTERFACE

// ---- mobject-server/_Internal/ChunkedRequests/HeaderAccessor/I_ChunkedRequestsHeaderAccessor.TcIO
INTERFACE I_ChunkedRequestsHeaderAccessor

METHOD PUBLIC TryGetChunkSequenceFromRequest : BOOL
VAR_INPUT
	Request : I_Request;
	Destination : REFERENCE TO DINT;
END_VAR
END_METHOD

METHOD PUBLIC TryGetChunkTotalFromRequest : BOOL
VAR_INPUT
	Request : I_Request;
	Destination : REFERENCE TO DINT;
END_VAR
END_METHOD

METHOD PUBLIC TryGetHasMoreChunksFromRequest : BOOL
VAR_INPUT
	Request : I_Request;
	Destination : REFERENCE TO BOOL;
END_VAR
END_METHOD

METHOD PUBLIC TryGetRequestIdFromRequest : BOOL
VAR_INPUT
	Request : I_Request;
	Destination : REFERENCE TO T_MAXSTRING;
END_VAR
END_METHOD

METHOD PUBLIC TryGetSessionIdFromRequest : BOOL
VAR_INPUT
	Request : I_Request;
	Destination : REFERENCE TO T_MAXSTRING;
END_VAR
END_METHOD

END_INTERFACE

// ---- mobject-server/_Internal/ChunkedRequests/Manager/I_ChunkedRequestsManager.TcIO
INTERFACE I_ChunkedRequestsManager

METHOD PUBLIC TryHandleIncomingRequest : BOOL
VAR_INPUT
	Request : I_Request;
	Response : I_ServerResponse;
	NextMidleware : I_Middleware;
END_VAR
END_METHOD

END_INTERFACE

// ---- mobject-server/_Internal/ChunkedRequests/SessionData/I_ChunkedRequestData.TcIO
INTERFACE I_ChunkedRequestData EXTENDS I_SessionData

PROPERTY PUBLIC IsComplete : BOOL
GET
END_GET
END_PROPERTY

PROPERTY PUBLIC PayloadAddress : POINTER TO STRING
GET
END_GET
END_PROPERTY

PROPERTY PUBLIC PayloadSizeInBytes : UDINT
GET
END_GET
END_PROPERTY

METHOD PUBLIC TryAddChunkedPayload : BOOL;
VAR_INPUT
	PayloadAddress : POINTER TO STRING;
	PayloadSize : UDINT;
	ChunkSequence : DINT;
END_VAR
END_METHOD

END_INTERFACE

// ---- mobject-server/_Internal/ChunkedResponses/HeaderAccessor/I_ChunkedResponseHeaderAccessor.TcIO
INTERFACE I_ChunkedResponseHeaderAccessor

METHOD PUBLIC TryGetResponseIdFromRequest : BOOL
VAR_INPUT
	Request : I_Request;
	Destination : ANY;
END_VAR
END_METHOD

METHOD PUBLIC TryGetSessionIdFromRequest : BOOL
VAR_INPUT
	Request : I_Request;
	Destination : REFERENCE TO T_MAXSTRING;
END_VAR
END_METHOD

METHOD PUBLIC TryGetSessionIdFromResponse : BOOL
VAR_INPUT
	Response : I_ServerResponse;
	Destination : ANY;
END_VAR
END_METHOD

METHOD PUBLIC UpdateResponseWithHasMoreChunks
VAR_INPUT
	Response : I_ServerResponse;
	ResponseId : T_MAXSTRING;
END_VAR
END_METHOD

END_INTERFACE

// ---- mobject-server/_Internal/ChunkedResponses/Manager/I_ChunkedResponseManager.TcIO
INTERFACE I_ChunkedResponseManager

METHOD PUBLIC HandleSuccessWithPayload;
VAR_INPUT
	OriginalResponse : I_ServerResponse;
	SourceAddress : PVOID;
	SourceSize : UDINT;
END_VAR
END_METHOD

METHOD PUBLIC TryHandleIncomingRequest : BOOL
VAR_INPUT
	Request : I_Request;
	Response : I_ServerResponse;
END_VAR
END_METHOD

END_INTERFACE

// ---- mobject-server/_Internal/ChunkedResponses/SessionData/I_ChunkedResponseData.TcIO
INTERFACE I_ChunkedResponseData EXTENDS I_SessionData

PROPERTY PUBLIC SendComplete : BOOL
GET
END_GET
END_PROPERTY

METHOD PUBLIC SendNextChunk
VAR_INPUT
	Response : I_ServerResponse;
	Size : UDINT;
END_VAR
END_METHOD

PROPERTY SizeRemaining : UDINT
GET
END_GET
END_PROPERTY

END_INTERFACE

// ---- mobject-server/_Internal/Header/I_Header.TcIO
INTERFACE I_Header

METHOD PUBLIC ToString
VAR_INPUT
	Destination : REFERENCE TO STRING(ServerConfiguration.HEADER_STRING_SIZE);
END_VAR
END_METHOD

METHOD PUBLIC TryGetField : BOOL;
VAR_INPUT
	Key : STRING;
	Destination : ANY;
END_VAR
END_METHOD

METHOD PUBLIC TryWriteField : BOOL;
VAR_INPUT
	Key : STRING;
	Source : ANY;
END_VAR
END_METHOD

END_INTERFACE

// ---- mobject-server/_Internal/Middleware/Interface/I_Middleware.TcIO
INTERFACE I_Middleware

METHOD Handle
VAR_INPUT
	Request : I_Request;
	Response : I_ServerResponse;
END_VAR
END_METHOD

PROPERTY PUBLIC NextMiddleware : I_Middleware
GET
END_GET
SET
END_SET
END_PROPERTY

END_INTERFACE

// ---- mobject-server/_Internal/Request/Interface/I_Request.TcIO
INTERFACE I_Request EXTENDS I_Disposable

PROPERTY PUBLIC CreatedTimestamp : I_Timestamp
GET
END_GET
END_PROPERTY

PROPERTY PUBLIC Header : I_Header
GET
END_GET
END_PROPERTY

PROPERTY PUBLIC PayloadAddress : POINTER TO STRING
GET
END_GET
END_PROPERTY

PROPERTY PUBLIC PayloadSizeInBytes : UDINT
GET
END_GET
END_PROPERTY

END_INTERFACE

// ---- mobject-server/_Internal/ResponseId/Interface/I_ResponseIdGenerator.TcIO
INTERFACE I_ResponseIdGenerator

METHOD PUBLIC Generate : T_MAXSTRING
VAR_INPUT
END_VAR
END_METHOD

END_INTERFACE

// ---- mobject-server/_Internal/RPC/AsyncRpcCallQueue/I_AsyncRpcCallQueue.TcIO
INTERFACE I_AsyncRpcCallQueue

METHOD PUBLIC TryAddRpcCall : BOOL
VAR_INPUT
	CallingParameters : I_Deserializer;
	CallingAsynchronousRpcResponse : I_AsynchronousRpcResponse;
	CallingHandler : I_AsynchronousRpcHandler;
END_VAR
END_METHOD

END_INTERFACE

// ---- mobject-server/_Internal/RPC/AsyncRpcCall/I_AsyncRpcCall.TcIO
INTERFACE I_AsyncRpcCall EXTENDS I_Disposable

METHOD PUBLIC Call
VAR_INPUT
END_VAR
END_METHOD

END_INTERFACE

// ---- mobject-server/_Internal/RPC/Handlers/I_AsynchronousRpcHandlers.TcIO
INTERFACE I_AsynchronousRpcHandlers

PROPERTY PUBLIC HasHandlers : BOOL
GET
END_GET
END_PROPERTY

METHOD PUBLIC TryGetByMethodName : BOOL
VAR_INPUT
	MethodName : T_MAXSTRING;
	Destination : REFERENCE TO I_AsynchronousRpcHandler;
END_VAR
END_METHOD

END_INTERFACE

// ---- mobject-server/_Internal/RPC/Handlers/I_HostAsynchronousRpcHandlers.TcIO
INTERFACE I_HostAsynchronousRpcHandlers

METHOD PUBLIC RegisterHandler
VAR_INPUT
	MethodName : T_MAXSTRING;
	Handler : I_AsynchronousRpcHandler;
END_VAR
END_METHOD

END_INTERFACE

// ---- mobject-server/_Internal/RPC/Handlers/I_HostSynchronousRpcHandlers.TcIO
INTERFACE I_HostSynchronousRpcHandlers

METHOD PUBLIC RegisterHandler
VAR_INPUT
	MethodName : T_MAXSTRING;
	Handler : I_SynchronousRpcHandler;
END_VAR
END_METHOD

END_INTERFACE

// ---- mobject-server/_Internal/RPC/Handlers/I_SynchronousRpcHandlers.TcIO
INTERFACE I_SynchronousRpcHandlers

PROPERTY PUBLIC HasHandlers : BOOL
GET
END_GET
END_PROPERTY

METHOD PUBLIC TryGetByMethodName : BOOL
VAR_INPUT
	MethodName : T_MAXSTRING;
	Destination : REFERENCE TO I_SynchronousRpcHandler;
END_VAR
END_METHOD

END_INTERFACE

// ---- mobject-server/_Internal/RPC/HeaderAccessor/I_RpcHeaderAccessor.TcIO
INTERFACE I_RpcHeaderAccessor

PROPERTY PUBLIC ContentType_Json : T_MAXSTRING
GET
END_GET
END_PROPERTY

METHOD PUBLIC TryGetAcceptResponseFormatFromRequest : BOOL
VAR_INPUT
	Request : I_Request;
	Destination : ANY;
END_VAR
END_METHOD

METHOD PUBLIC TryGetContentTypeFromRequest : BOOL
VAR_INPUT
	Request : I_Request;
	Destination : ANY;
END_VAR
END_METHOD

METHOD PUBLIC TryGetMethodNameFromRequest : BOOL
VAR_INPUT
	Request : I_Request;
	Destination : ANY;
END_VAR
END_METHOD

METHOD PUBLIC TryGetTypeFromRequest : BOOL
VAR_INPUT
	Request : I_Request;
	Destination : ANY;
END_VAR
END_METHOD

END_INTERFACE

// ---- mobject-server/_Internal/RPC/Manager/I_RpcManager.TcIO
INTERFACE I_RpcManager

METHOD PUBLIC TryHandleIncomingRequest : BOOL
VAR_INPUT
	Request : I_Request;
	Response : I_ServerResponse;
END_VAR
END_METHOD

END_INTERFACE

// ---- mobject-server/_Internal/RPC/Response/Async/I_AsynchronousRpcResponse.TcIO
INTERFACE I_AsynchronousRpcResponse EXTENDS I_Disposable

METHOD PUBLIC CompleteWithBase64
VAR_INPUT
	pBytes : POINTER TO BYTE;
	nBytes : DINT;
END_VAR
END_METHOD

METHOD PUBLIC CompleteWithBool
VAR_INPUT
	Value : BOOL;
END_VAR
END_METHOD

METHOD PUBLIC CompleteWithBytesAsHex
VAR_INPUT
	pBytes : POINTER TO BYTE;
	nBytes : DINT;
END_VAR
END_METHOD

METHOD PUBLIC CompleteWithDateTime
VAR_INPUT
	Value : DATE_AND_TIME;
END_VAR
END_METHOD

METHOD PUBLIC CompleteWithDcTime
VAR_INPUT
	Value : DCTIME;
END_VAR
END_METHOD

METHOD PUBLIC CompleteWithDint
VAR_INPUT
	Value : DINT;
END_VAR
END_METHOD

METHOD PUBLIC CompleteWithFileTime
VAR_INPUT
	Value : FILETIME;
END_VAR
END_METHOD

METHOD PUBLIC CompleteWithLint
VAR_INPUT
	Value : LINT;
END_VAR
END_METHOD

METHOD PUBLIC CompleteWithLreal
VAR_INPUT
	Value : LREAL;
END_VAR
END_METHOD

METHOD PUBLIC CompleteWithNull
VAR_INPUT
END_VAR
END_METHOD

METHOD PUBLIC CompleteWithObject
VAR_INPUT
	Object : I_Serializable;
END_VAR
END_METHOD

METHOD PUBLIC CompleteWithReal
VAR_INPUT
	Value : REAL;
END_VAR
END_METHOD

METHOD PUBLIC CompleteWithSerializer
VAR_INPUT
	Serializer : I_Serializer;
END_VAR
END_METHOD

METHOD PUBLIC CompleteWithString
VAR_INPUT
	Value : T_MAXSTRING;
END_VAR
END_METHOD

METHOD PUBLIC CompleteWithUdint
VAR_INPUT
	Value : UDINT;
END_VAR
END_METHOD

METHOD PUBLIC CompleteWithUlint
VAR_INPUT
	Value : ULINT;
END_VAR
END_METHOD

METHOD PUBLIC GetSerializer : I_Serializer
VAR_INPUT
END_VAR
END_METHOD

METHOD PUBLIC RejectWithError
VAR_INPUT
	ErrorCode : T_MAXSTRING;
	Message : T_MAXSTRING;
END_VAR
END_METHOD

END_INTERFACE

// ---- mobject-server/_Internal/RPC/Response/Factory/I_AsynchronousRpcResponseFactory.TcIO
INTERFACE I_AsynchronousRpcResponseFactory

METHOD PUBLIC TryCreate : BOOL
VAR_INPUT
	Destination : REFERENCE TO I_AsynchronousRpcResponse;
END_VAR
END_METHOD

END_INTERFACE

// ---- mobject-server/_Internal/RPC/Response/Sync/I_SynchronousRpcResponse.TcIO
INTERFACE I_SynchronousRpcResponse EXTENDS I_Disposable

METHOD PUBLIC CompleteWithBase64
VAR_INPUT
	pBytes : POINTER TO BYTE;
	nBytes : DINT;
END_VAR
END_METHOD

METHOD PUBLIC CompleteWithBool
VAR_INPUT
	Value : BOOL;
END_VAR
END_METHOD

METHOD PUBLIC CompleteWithBytesAsHex
VAR_INPUT
	pBytes : POINTER TO BYTE;
	nBytes : DINT;
END_VAR
END_METHOD

METHOD PUBLIC CompleteWithDateTime
VAR_INPUT
	Value : DATE_AND_TIME;
END_VAR
END_METHOD

METHOD PUBLIC CompleteWithDcTime
VAR_INPUT
	Value : DCTIME;
END_VAR
END_METHOD

METHOD PUBLIC CompleteWithDint
VAR_INPUT
	Value : DINT;
END_VAR
END_METHOD

METHOD PUBLIC CompleteWithFileTime
VAR_INPUT
	Value : FILETIME;
END_VAR
END_METHOD

METHOD PUBLIC CompleteWithLint
VAR_INPUT
	Value : LINT;
END_VAR
END_METHOD

METHOD PUBLIC CompleteWithLreal
VAR_INPUT
	Value : LREAL;
END_VAR
END_METHOD

METHOD PUBLIC CompleteWithNull
VAR_INPUT
END_VAR
END_METHOD

METHOD PUBLIC CompleteWithObject
VAR_INPUT
	Object : I_Serializable;
END_VAR
END_METHOD

METHOD PUBLIC CompleteWithReal
VAR_INPUT
	Value : REAL;
END_VAR
END_METHOD

METHOD PUBLIC CompleteWithSerializer
VAR_INPUT
	Serializer : I_Serializer;
END_VAR
END_METHOD

METHOD PUBLIC CompleteWithString
VAR_INPUT
	Value : T_MAXSTRING;
END_VAR
END_METHOD

METHOD PUBLIC CompleteWithUdint
VAR_INPUT
	Value : UDINT;
END_VAR
END_METHOD

METHOD PUBLIC CompleteWithUlint
VAR_INPUT
	Value : ULINT;
END_VAR
END_METHOD

METHOD PUBLIC GetSerializer : I_Serializer
VAR_INPUT
END_VAR
END_METHOD

METHOD PUBLIC RejectWithError
VAR_INPUT
	ErrorCode : T_MAXSTRING;
	Message : T_MAXSTRING;
END_VAR
END_METHOD

METHOD PUBLIC TryMakeAsynchronous : BOOL
VAR_INPUT
	Destination : REFERENCE TO I_AsynchronousRpcResponse;
END_VAR
END_METHOD

END_INTERFACE

// ---- mobject-server/_Internal/ServerResponse/HeaderAccessor/I_ServerResponseHeaderAccessor.TcIO
INTERFACE I_ServerResponseHeaderAccessor

METHOD PUBLIC UpdateResponseWithAccepted
VAR_INPUT
	Response : I_ServerResponse;
END_VAR
END_METHOD

METHOD PUBLIC UpdateResponseWithBusy
VAR_INPUT
	Response : I_ServerResponse;
END_VAR
END_METHOD

METHOD PUBLIC UpdateResponseWithError
VAR_INPUT
	Response : I_ServerResponse;
	ErrorCode : T_MAXSTRING;
	Message : T_MAXSTRING;
END_VAR
END_METHOD

METHOD PUBLIC UpdateResponseWithPending
VAR_INPUT
	Response : I_ServerResponse;
	ResponseId : T_MAXSTRING;
	RetryDelayInMs : UDINT;
END_VAR
END_METHOD

METHOD PUBLIC UpdateResponseWithSuccess
VAR_INPUT
	Response : I_ServerResponse;
END_VAR
END_METHOD

END_INTERFACE

// ---- mobject-server/_Internal/ServerResponse/Interface/I_ServerResponse.TcIO
INTERFACE I_ServerResponse

METHOD PUBLIC Accepted
VAR_INPUT
END_VAR
END_METHOD

METHOD PUBLIC Busy
VAR_INPUT
END_VAR
END_METHOD

METHOD PUBLIC Error
VAR_INPUT
	ErrorCode : T_MAXSTRING;
	Message : T_MAXSTRING;
END_VAR
END_METHOD

PROPERTY PUBLIC Header : I_Header
GET
END_GET
END_PROPERTY

PROPERTY PUBLIC HeadersSent : BOOL
GET
END_GET
END_PROPERTY

METHOD PUBLIC Pending
VAR_INPUT
	ResponseId : REFERENCE TO T_MAXSTRING;
	RetryDelayInMs : UDINT;
END_VAR
END_METHOD

METHOD PUBLIC Success
VAR_INPUT
END_VAR
END_METHOD

METHOD PUBLIC SuccessWithPayload
VAR_INPUT
	PayloadDataAddress : PVOID;
	
	// Number of payload bytes to copy.
    // Does not include the STRING null terminator.
	PayloadDataSize : UDINT;
END_VAR
END_METHOD

END_INTERFACE

// ---- mobject-server/_Internal/Sessions/HeaderAccessor/I_SessionHeaderAccessor.TcIO
INTERFACE I_SessionHeaderAccessor

METHOD PUBLIC TryGetResponseIdFromRequest : BOOL
VAR_INPUT
	Request : I_Request;
	Destination : ANY;
END_VAR
END_METHOD

METHOD PUBLIC TryGetSessionIdFromRequest : BOOL
VAR_INPUT
	Request : I_Request;
	Destination : REFERENCE TO T_MAXSTRING;
END_VAR
END_METHOD

METHOD PUBLIC UpdateRequestWithSessionId
VAR_INPUT
	Request : I_Request;
	SessionId : T_MAXSTRING;
END_VAR
END_METHOD

METHOD PUBLIC UpdateResponseWithSessionId
VAR_INPUT
	Response : I_ServerResponse;
	SessionId : T_MAXSTRING;
END_VAR
END_METHOD

END_INTERFACE

// ---- mobject-server/_Internal/Sessions/Manager/I_SessionManager.TcIO
INTERFACE I_SessionManager

METHOD PUBLIC CreateSession : T_MAXSTRING
END_METHOD

METHOD PUBLIC DisposeAllSessions
VAR_INPUT
END_VAR
END_METHOD

METHOD PUBLIC IsValidSession : BOOL
VAR_INPUT
	Id : T_MAXSTRING;
END_VAR
END_METHOD

METHOD PUBLIC RefreshSession
VAR_INPUT
	Id : T_MAXSTRING;
END_VAR
END_METHOD

END_INTERFACE

// ---- mobject-server/_Internal/Sessions/SessionData/I_SessionData.TcIO
INTERFACE I_SessionData EXTENDS I_Disposable

END_INTERFACE

// ---- mobject-server/_Internal/Sessions/SessionId/I_SessionIdGenerator.TcIO
INTERFACE I_SessionIdGenerator

METHOD PUBLIC Generate : T_MAXSTRING
VAR_INPUT
END_VAR
END_METHOD

END_INTERFACE

// ---- mobject-server/_Internal/Sessions/Session/I_Session.TcIO
INTERFACE I_Session Extends I_Disposable

METHOD PUBLIC AddOrUpdateStorage
VAR_INPUT
	StorageId : T_MAXSTRING;
	Source : I_SessionData;
END_VAR
END_METHOD

METHOD PUBLIC DisposeAllDataFromStorage
VAR_INPUT
END_VAR
END_METHOD

METHOD PUBLIC DisposeDataFromStorage
VAR_INPUT
	StorageId : T_MAXSTRING;
END_VAR
END_METHOD

PROPERTY PUBLIC Id : T_MAXSTRING
GET
END_GET
END_PROPERTY

PROPERTY PUBLIC LastAccessedTimestamp : I_TimeStamp
GET
END_GET
END_PROPERTY

METHOD PUBLIC Refresh
VAR_INPUT
END_VAR
END_METHOD

METHOD PUBLIC TryGetDataFromStorage : BOOL
VAR_INPUT
	StorageId : T_MAXSTRING;
	Destination : REFERENCE TO I_SessionData;
END_VAR
END_METHOD

END_INTERFACE

// ---- mobject-server/_Internal/Sessions/Storage/I_SessionStorage.TcIO
INTERFACE I_SessionStorage

METHOD PUBLIC DisposeSessionDataById
VAR_INPUT
	SessionId : T_MAXSTRING;
	StorageId : T_MAXSTRING;
END_VAR
END_METHOD

METHOD PUBLIC TryRetrieveSessionDataById : BOOL
VAR_INPUT
	SessionId : T_MAXSTRING;
	StorageId : T_MAXSTRING;
	Destination : REFERENCE TO I_SessionData;
END_VAR
END_METHOD

METHOD PUBLIC TryStoreSessionDataById : BOOL
VAR_INPUT
	SessionId : T_MAXSTRING;
	StorageId : T_MAXSTRING;
	Source : I_SessionData;
END_VAR
END_METHOD

END_INTERFACE

// ---- mobject-server/_Internal/TimeStamp/I_Timestamp.TcIO
INTERFACE I_Timestamp

METHOD PUBLIC IsDurationElapsed : BOOL
VAR_INPUT
	Duration : TIME;
END_VAR
END_METHOD

PROPERTY PUBLIC TimeSince : TIME
GET
END_GET
END_PROPERTY

END_INTERFACE

// ---- mobject-collections/Dictionary/Dictionary.TcPOU
{attribute 'linkalways'} 
{attribute 'no_explicit_call' := 'This FB is a CLASS and must be accessed using methods or properties'}
{attribute 'enable_dynamic_creation'}
FUNCTION_BLOCK Dictionary EXTENDS Disposable IMPLEMENTS I_Dictionary
VAR
	eventEmitter : EventEmitter;
	rootNode : I_DictionaryTreeNode;
END_VAR

METHOD PUBLIC AddOrUpdate
VAR_INPUT
	Key : T_MAXSTRING;
	Value : ANY;
END_VAR
rootNode := THIS^.RecursiveInsert(Key, Value, rootNode);
EmitChangedEvent();
END_METHOD

METHOD PRIVATE Balance : I_DictionaryTreeNode
VAR_INPUT
	Node : I_DictionaryTreeNode;
END_VAR
VAR
	balanceFactor : DINT;
END_VAR
balanceFactor := THIS^.GetBalanceFactor(Node);

IF (balanceFactor > 1) THEN
	IF THIS^.GetBalanceFactor(Node.Left) < 0 THEN
		Node.Left := THIS^.LeftRotate(Node.Left);
	END_IF
	Node := RightRotate(Node);
ELSIF (balanceFactor < -1) THEN
	IF THIS^.GetBalanceFactor(Node.Right) > 0 THEN
		Node.Right := RightRotate(Node.Right);
	END_IF
	Node := LeftRotate(Node);
END_IF

Balance := Node;
END_METHOD

METHOD PUBLIC Clear
VAR_INPUT
END_VAR
IF rootNode = 0 THEN
	RETURN;
END_IF

THIS^.RecursiveClear(rootNode);
rootNode := 0;
EmitChangedEvent();
END_METHOD

METHOD PUBLIC ContainsKey : BOOL
VAR_INPUT
	Key : T_MAXSTRING;
END_VAR
VAR
	foundNode : I_DictionaryTreeNode;
END_VAR
foundNode := THIS^.RecursiveFind(Key, rootNode);

IF foundNode = 0 THEN
	RETURN;
END_IF

ContainsKey := TRUE;
END_METHOD

PROPERTY PUBLIC Count : DINT
GET
VAR
	NodeCount : DINT;
END_VAR
RecursiveCountNodes(rootNode, NodeCount);
Count := NodeCount;
END_GET
END_PROPERTY

METHOD PRIVATE EmitChangedEvent
VAR
	pDictionaryChangedEvent : POINTER TO KeyValueCollectionChangedEvent;
END_VAR
pDictionaryChangedEvent := __NEW(KeyValueCollectionChangedEvent(Target := THIS^));
eventEmitter.Emit('OnChanged', pDictionaryChangedEvent^);
pDictionaryChangedEvent^.Dispose();
END_METHOD

METHOD PRIVATE EmitDisposedEvent
VAR
	pDictionaryDisposedEvent : POINTER TO KeyValueCollectionDisposedEvent;
END_VAR
pDictionaryDisposedEvent := __NEW(KeyValueCollectionDisposedEvent(Target := THIS^));
eventEmitter.Emit('OnDisposed', pDictionaryDisposedEvent^);
pDictionaryDisposedEvent^.Dispose();
END_METHOD

METHOD FB_exit : BOOL
VAR_INPUT
	bInCopyCode : BOOL; // if TRUE, the exit method is called for exiting an instance that is copied afterwards (online change).
END_VAR
VAR
END_VAR
IF bInCopyCode THEN
    RETURN;
END_IF

Clear();
EmitDisposedEvent();
END_METHOD

METHOD PRIVATE FindMinimum : I_DictionaryTreeNode
VAR_INPUT
	Node : I_DictionaryTreeNode;
END_VAR
VAR
	nextNode : I_DictionaryTreeNode;
END_VAR
nextNode := Node;

WHILE (nextNode.left <> 0) DO
      nextNode := nextNode.left;
END_WHILE;

FindMinimum := nextNode;
END_METHOD

METHOD PRIVATE GetBalanceFactor : DINT
VAR_INPUT
	Node : I_DictionaryTreeNode;
END_VAR
IF (Node = 0) THEN
	GetBalanceFactor := 0;
	RETURN;
END_IF

GetBalanceFactor := THIS^.GetHeight(node.left) - THIS^.GetHeight(node.right);
END_METHOD

METHOD GetEnumerator : I_ForwardEnumerator
VAR
	pNodeCollection : POINTER TO LinkedList;
	pEnumerator : POINTER TO DictionaryForwardEnumerator;
END_VAR
pNodeCollection := __NEW(LinkedList);
THIS^.RecursiveAddNodesInOrderToCollection(rootNode, pNodeCollection^);

pEnumerator := __NEW(DictionaryForwardEnumerator(Parent := THIS^, Nodes := pNodeCollection^));
GetEnumerator := pEnumerator^;
END_METHOD

METHOD PRIVATE GetHeight : DINT
VAR_INPUT
	Node : I_DictionaryTreeNode;
END_VAR
IF Node = 0 THEN
	GetHeight := -1;
	RETURN;
END_IF

GetHeight := Node.Height;
END_METHOD

METHOD PUBLIC GetKeys : I_Collection
VAR
	pLinkedList : POINTER TO LinkedList;
END_VAR
pLinkedList := __NEW(LinkedList);
THIS^.RecursiveAddKeysInOrderToCollection(rootNode,pLinkedList^);
GetKeys := pLinkedList^;
END_METHOD

METHOD GetKeyValueEnumerator : I_KeyValueForwardEnumerator
VAR
	pNodeCollection : POINTER TO LinkedList;
	pEnumerator : POINTER TO DictionaryForwardEnumerator;
END_VAR
pNodeCollection := __NEW(LinkedList);
THIS^.RecursiveAddNodesInOrderToCollection(rootNode, pNodeCollection^);

pEnumerator := __NEW(DictionaryForwardEnumerator(Parent := THIS^, Nodes := pNodeCollection^));
GetKeyValueEnumerator := pEnumerator^;
END_METHOD

PROPERTY IsEmpty : BOOL
GET
IsEmpty := rootNode = 0;
END_GET
END_PROPERTY

METHOD PRIVATE LeftRotate : I_DictionaryTreeNode
VAR_INPUT
	X : I_DictionaryTreeNode;
END_VAR
VAR
	y : I_DictionaryTreeNode;
	t2 : I_DictionaryTreeNode;
END_VAR
y := X.right;
t2 := y.left;
y.left := X;
X.right := t2;
THIS^.UpdateHeight(X);
THIS^.UpdateHeight(y);
LeftRotate := y;
END_METHOD

METHOD PUBLIC OffEvent
VAR_INPUT
	EventName : T_MaxString;
	EventHandler : I_EventHandler;
END_VAR
eventEmitter.OffEvent(EventName, EventHandler);
END_METHOD

METHOD PUBLIC OnceEvent
VAR_INPUT
	EventName : T_MaxString;
	EventHandler : I_EventHandler;
END_VAR
eventEmitter.OnceEvent(EventName, EventHandler);
END_METHOD

METHOD PUBLIC OnEvent
VAR_INPUT
	EventName : T_MaxString;
	EventHandler : I_EventHandler;
END_VAR
eventEmitter.OnEvent(EventName, EventHandler);
END_METHOD

METHOD PRIVATE RecursiveAddKeysInOrderToCollection
VAR_INPUT
	Node : I_DictionaryTreeNode;
	Collection : I_Collection;
END_VAR
VAR
	key : T_MAXSTRING;
END_VAR
IF Node = 0 THEN
	RETURN;
END_IF

THIS^.RecursiveAddKeysInOrderToCollection(Node.Left,Collection);
key := Node.Key;
Collection.AddItem(key);
THIS^.RecursiveAddKeysInOrderToCollection(Node.Right,Collection);
END_METHOD

METHOD PRIVATE RecursiveAddNodesInOrderToCollection
VAR_INPUT
	Node : I_DictionaryTreeNode;
	Collection : I_Collection;
END_VAR
IF Node = 0 THEN
	RETURN;
END_IF

THIS^.RecursiveAddNodesInOrderToCollection(Node.Left,Collection);
Collection.AddItem(Node);
THIS^.RecursiveAddNodesInOrderToCollection(Node.Right,Collection);
END_METHOD

METHOD PRIVATE RecursiveClear
VAR_INPUT
	Node : I_DictionaryTreeNode;
END_VAR
VAR
	thisNodeKey : T_MAXSTRING;
	leftNodeKey : T_MAXSTRING;
	rightNodeKey : T_MAXSTRING;
END_VAR
IF (Node = 0) THEN
	RETURN;
END_IF

thisNodeKey := Node.key;

IF (Node.Left <> 0) THEN
	leftNodeKey := Node.Left.key;
END_IF

IF (Node.Right <> 0) THEN
	rightNodeKey := Node.Right.key;
END_IF


RecursiveClear(Node.Left);
RecursiveClear(Node.Right);
Node.Dispose();
END_METHOD

METHOD PRIVATE RecursiveCountNodes
VAR_INPUT
	Node : I_DictionaryTreeNode;
	Count : REFERENCE TO DINT;
END_VAR
IF Node = 0 THEN
	RETURN;
END_IF

Count := Count + 1;

THIS^.RecursiveCountNodes(Node.Left,Count);
THIS^.RecursiveCountNodes(Node.Right,Count);
END_METHOD

METHOD PRIVATE RecursiveDelete : I_DictionaryTreeNode
VAR_INPUT
	Key : T_MAXSTRING;
	Node : I_DictionaryTreeNode;
END_VAR
VAR
	newNode : I_DictionaryTreeNode; 
	minValueNode : I_DictionaryTreeNode;
	minValueNodeParent : I_DictionaryTreeNode;
	balanceFactor : DINT;
END_VAR
IF (Node = 0) THEN
    RETURN;
END_IF

IF (Key < Node.Key) THEN
    Node.left := THIS^.RecursiveDelete(Key, Node.left);
ELSIF (Key > Node.Key) THEN
    Node.right := THIS^.RecursiveDelete(Key, Node.right);
ELSE
    IF (Node.Left = 0) OR (Node.Right = 0) THEN
        IF (Node.Left = 0) THEN
            newNode := Node.Right;
        ELSE
            newNode := Node.Left;
        END_IF

        Node.Dispose();
        THIS^.updateHeight(newNode);
        RecursiveDelete := THIS^.Balance(newNode);
        RETURN;
    ELSE
        minValueNode := FindMinimum(Node.Right);
        Node.DeepCopy(minValueNode);
        Node.Right := THIS^.RecursiveDelete(minValueNode.Key, Node.Right);	
    END_IF
END_IF

THIS^.updateHeight(Node);
RecursiveDelete := THIS^.Balance(Node);
END_METHOD

METHOD PRIVATE RecursiveFind : I_DictionaryTreeNode
VAR_INPUT
	Key : T_MAXSTRING;
	Node : I_DictionaryTreeNode;
END_VAR
IF (Node = 0) THEN
	RETURN;
END_IF

IF (Key < Node.key) THEN
  RecursiveFind := THIS^.RecursiveFind(key, Node.left);
  RETURN;
ELSIF (key > Node.key) THEN
  RecursiveFind := THIS^.RecursiveFind(key, Node.right);
  RETURN;
ELSE 
  RecursiveFind := Node;
  RETURN;
END_IF
END_METHOD

METHOD PRIVATE RecursiveInsert : I_DictionaryTreeNode
VAR_INPUT
	Key : T_MAXSTRING;
	Value : ANY;
	Node : I_DictionaryTreeNode;
END_VAR
VAR
	pAVLTreeNode : POINTER TO DictionaryTreeNode;
	balanceFactor : DINT;
END_VAR
IF (Node = 0) THEN
	pAVLTreeNode := __NEW(DictionaryTreeNode(NodeKey := Key, NodeSource := Value));
	RecursiveInsert := pAVLTreeNode^;
	RETURN;
END_IF

IF (Key < Node.Key) THEN
	Node.left := THIS^.RecursiveInsert(Key, Value, Node.left);
ELSIF (Key > Node.Key) THEN
	Node.right := THIS^.RecursiveInsert(Key, Value, Node.right);
ELSE
	Node.Reinitialize(Key,Value);
	RecursiveInsert := Node;
END_IF

THIS^.updateHeight(node);

Node := balance(Node);
RecursiveInsert := Node;
END_METHOD

METHOD PUBLIC Remove
VAR_INPUT
	Key : T_MAXSTRING;
END_VAR
rootNode := THIS^.RecursiveDelete(Key, rootNode);
EmitChangedEvent();
END_METHOD

METHOD PRIVATE RightRotate : I_DictionaryTreeNode
VAR_INPUT
	Y : I_DictionaryTreeNode;
END_VAR
VAR
	x : I_DictionaryTreeNode;
	t2 : I_DictionaryTreeNode;
END_VAR
x := Y.left;
t2 := x.right;
x.right := Y;
Y.left := t2;
THIS^.UpdateHeight(Y);
THIS^.UpdateHeight(x);
RightRotate := x;
END_METHOD

METHOD PUBLIC TryAdd : BOOL
VAR_INPUT
	Key : T_MAXSTRING;
	Value : ANY;
END_VAR
IF ContainsKey(Key) THEN
	RETURN;
END_IF
	  
THIS^.AddOrUpdate(Key, Value);
TryAdd := TRUE;
END_METHOD

METHOD PUBLIC TryGetValue : BOOL
VAR_INPUT
	Key : T_MAXSTRING;
	Destination	: ANY;
END_VAR
TryGetValue := TryGetValueTo(Key, Destination.pValue, DINT_TO_UDINT(Destination.diSize));
END_METHOD

METHOD PUBLIC TryGetValueTo : BOOL
VAR_INPUT
	Key : T_MAXSTRING;
	DestinationAddress : PVOID;
	DestinationSize : UDINT;
END_VAR
VAR
	foundNode : I_DictionaryTreeNode;
END_VAR
foundNode := THIS^.RecursiveFind(Key, rootNode);

IF foundNode = 0 THEN
	RETURN;
END_IF

TryGetValueTo := foundNode.TryGetTo(DestinationAddress, DestinationSize);
END_METHOD

METHOD PRIVATE UpdateHeight
VAR_INPUT
	Node : I_DictionaryTreeNode;
END_VAR
IF (Node = 0) THEN
	RETURN;
END_IF

Node.height := 1 + MAX(THIS^.GetHeight(Node.left), THIS^.GetHeight(Node.right));
END_METHOD

END_FUNCTION_BLOCK

// ---- mobject-collections/OrderedDictionary/OrderedDictionary.TcPOU
{attribute 'linkalways'} 
{attribute 'no_explicit_call' := 'This FB is a CLASS and must be accessed using methods or properties'}
{attribute 'enable_dynamic_creation'}
FUNCTION_BLOCK OrderedDictionary EXTENDS Disposable IMPLEMENTS I_Dictionary
VAR
	eventEmitter : EventEmitter;
	rootNode : I_OrderedDictionaryTreeNode;
	head : I_OrderedDictionaryTreeNode;
	tail : I_OrderedDictionaryTreeNode;
END_VAR

METHOD PRIVATE AddKeysInOrderToCollection
VAR_INPUT
	Collection : I_Collection;
END_VAR
VAR
	currentNode : I_OrderedDictionaryTreeNode;
	key : T_MAXSTRING;
END_VAR
IF head = 0 THEN
	RETURN;
END_IF

currentNode := head;

REPEAT
    key := currentNode.Key;
	Collection.AddItem(key);
	currentNode := currentNode.Next;
UNTIL
    currentNode = 0
END_REPEAT;
END_METHOD

METHOD PRIVATE AddNodesInOrderToCollection
VAR_INPUT
	Collection : I_Collection;
END_VAR
VAR
	currentNode : I_OrderedDictionaryTreeNode;
	key : T_MAXSTRING;
END_VAR
IF head = 0 THEN
	RETURN;
END_IF

currentNode := head;

REPEAT
	Collection.AddItem(currentNode);
	currentNode := currentNode.Next;
UNTIL
    currentNode = 0
END_REPEAT;
END_METHOD

METHOD PRIVATE AddNodeToEnd
VAR_INPUT
	Node : I_OrderedDictionaryTreeNode;
END_VAR
VAR
	originalTailNode : I_OrderedDictionaryTreeNode;
END_VAR
//LogMsg_I_OrderedDictionaryTreeNode('OrderedDictionary', 'AddNodeToEnd: Called with', Node);

IF head = 0 THEN
	head := Node;
	tail := Node;
	Node.Previous := 0;
	Node.Next := 0;
//	LogMsg('OrderedDictionary', 'AddNodeToEnd: Return, head = 0');
//	LogMsg_I_OrderedDictionaryTreeNode('OrderedDictionary', 'AddNodeToEnd: Head is', head);
//	LogMsg_I_OrderedDictionaryTreeNode('OrderedDictionary', 'AddNodeToEnd: Tail is', tail);
	RETURN;
END_IF

//LogMsg_I_OrderedDictionaryTreeNode('OrderedDictionary', 'AddNodeToEnd: Original Tail was', tail);
originalTailNode := tail;
tail := Node;
//LogMsg_I_OrderedDictionaryTreeNode('OrderedDictionary', 'AddNodeToEnd: Tail is now', tail);

originalTailNode.Next := node;
//LogMsg_I_OrderedDictionaryTreeNode('OrderedDictionary', 'AddNodeToEnd: Original Tail next is', originalTailNode.Next);
tail.Previous := originalTailNode;
tail.Next := 0;
//LogMsg_I_OrderedDictionaryTreeNode('OrderedDictionary', 'AddNodeToEnd: Tail previous is now', tail.Previous);

//LogMsg('OrderedDictionary', 'AddNodeToEnd: Return');
END_METHOD

METHOD PUBLIC AddOrUpdate
VAR_INPUT
	Key : T_MAXSTRING;
	Value : ANY;
END_VAR
rootNode := THIS^.RecursiveInsert(Key, Value, rootNode);
EmitChangedEvent();
END_METHOD

